Yaskawa INFORM job: OK_R2_O8B-O21B(90,0)_MPKMOK.JBI

/JOB
//NAME OK_R2_O8B-O21B(90,0)_MPKMOK
///FOLDERNAME X4
//POS
///NPOS 666,666,666,28,0,0
///TOOL 0
///POSTYPE PULSE
///PULSE
C00000=91699,-114837,-126172,-5297,65572,-69852
C00001=92194,-112793,-113721,-5907,59024,-69345
C00002=110766,-104046,-107477,-16255,62170,-62558
C00003=110766,-104165,-106515,-16351,61543,-62463
C00004=110766,-104147,-106683,-16334,61651,-62479
C00005=111036,-99665,-105018,-16294,62933,-62564
C00006=110753,-104252,-107692,-16244,62194,-62563
C00007=67116,-81864,-100907,8307,67410,-78303
C00008=67696,-81353,-98479,8065,66136,-78195
C00009=67696,-81727,-97702,8106,65471,-78242
C00010=67696,-81654,-97861,8098,65606,-78232
C00011=68924,-78441,-96430,7380,66259,-77758
C00012=67562,-81507,-99004,8124,66390,-78224
C00013=94591,-107711,-114910,-7081,62535,-68652
C00014=75177,-96078,-118139,-30635,103857,57240
C00015=71016,-101172,-117038,-29652,99603,56842
C00016=69320,-102842,-116458,-29300,97976,56637
C00017=65815,-114376,-118551,-28520,92729,56653
C00018=65815,-114603,-117718,-28482,92175,56787
C00019=65333,-115185,-120736,-28492,93393,56311
C00020=69320,-102842,-116458,-29300,97976,56637
C00021=95416,-92028,-88987,-60066,102481,86035
C00022=94783,-95327,-90301,-59871,101628,86283
C00023=95175,-93300,-89498,-59989,102155,86131
C00024=95403,-90904,-93442,-60883,104178,84663
C00025=96846,-88575,-93381,-61258,105655,84430
C00026=100267,-82342,-92970,-62384,109223,83757
C00027=98853,-105972,-123361,-35115,85568,62201
C00028=123874,-116503,-132949,-35316,93358,57662
C00029=98784,-130821,-129289,-12660,72810,27269
C00030=95442,-119682,-123188,-11300,74256,25961
C00031=89918,-115832,-119261,-9213,73142,24151
C00032=89918,-116068,-118310,-9245,72445,24204
C00033=89918,-115832,-119261,-9213,73142,24151
C00034=86534,-112000,-117975,-7848,73961,22933
C00035=89918,-115832,-119261,-9213,73142,24151
C00036=91545,-105966,-115876,-9715,76271,24462
C00037=89918,-115832,-119261,-9213,73142,24151
C00038=100559,-101270,-121421,-12879,83175,26784
C00039=103898,-109015,-126857,-14089,83070,27872
C00040=112603,-104533,-117877,-29713,115926,66306
C00041=112603,-104533,-117877,-29713,115926,66306
C00042=102787,-102282,-117268,-28859,121596,74546
C00043=102787,-103288,-115881,-28417,120387,74903
C00044=102787,-102191,-117377,-28898,121696,74514
C00045=102247,-107992,-119426,-28435,120002,74778
C00046=104853,-110239,-121572,-27980,116786,76632
C00047=123177,-144145,-129947,-26642,102859,76425
C00048=123829,-162749,-132848,-26863,92935,75206
C00049=121638,-162916,-132889,-27033,92171,74551
C00050=123829,-165003,-135169,-26874,93176,75150
C00051=112500,-101779,-108680,-28673,112161,67324
C00052=131997,-56357,-109229,4920,90907,66095
C00053=147842,-82951,-112210,34984,98309,69155
C00054=149737,-87239,-109966,34223,94635,68708
C00055=151378,-90687,-107740,33690,91394,68340
C00056=151378,-91074,-107136,33673,90915,68196
C00057=151378,-90687,-107740,33690,91394,68340
C00058=145558,-100693,-110774,34812,90892,65938
C00059=145748,-102567,-109629,34742,89434,65557
C00060=146398,-106855,-111180,34614,88141,65411
C00061=145748,-102567,-109629,34742,89434,65557
C00062=144942,-96836,-108242,34942,91483,65883
C00063=124830,-105124,-96789,55472,88700,57654
C00064=126521,-104925,-96716,55344,87736,58010
C00065=123249,-105523,-98221,55595,90026,57599
C00066=144949,-101354,-110618,34915,90771,65662
C00067=150499,-88658,-108954,33966,93222,68562
C00068=149737,-87239,-109966,34223,94635,68708
C00069=147842,-82951,-112210,34984,98309,69155
C00070=134744,-82461,-113999,23220,99839,19223
C00071=107178,-113461,-99894,5964,101445,-70182
C00072=116777,-120475,-92303,7084,92443,-67341
C00073=117649,-121004,-89231,7177,90217,-67172
C00074=117541,-124461,-90223,7160,89070,-67274
C00075=117649,-121004,-89231,7177,90217,-67172
C00076=121247,-121045,-89244,7619,89875,-65972
C00077=117649,-121004,-89231,7177,90217,-67172
C00078=120454,-123758,-93756,7530,91322,-66155
C00079=131821,-147240,-100571,7170,74455,-63187
C00080=132564,-146887,-99168,7097,73320,-62988
C00081=132564,-147261,-99594,7095,73390,-62984
C00082=116129,-123152,-95240,7006,92928,-67534
C00083=114019,-118624,-94636,6761,95050,-68140
C00084=115483,-77500,-114184,-15325,109930,-22258
C00085=107117,-124945,-135933,21570,97656,-8797
C00086=118143,-111392,-129277,15030,88270,9704
C00087=118164,-109444,-128626,15025,88847,9780
C00088=118164,-110450,-128026,15024,87989,9675
C00089=118164,-110074,-128260,15024,88315,9716
C00090=118257,-101380,-125250,15013,90827,10051
C00091=118164,-108155,-129289,15031,89881,9907
C00092=110085,-126828,-135239,17345,85673,6704
C00093=92891,-111374,-130366,26323,94899,-34453
C00094=97190,-111538,-124535,25207,90331,-33950
C00095=98877,-113015,-125031,24804,89436,-33545
C00096=97190,-111538,-124535,25207,90331,-33950
C00097=97263,-106439,-128356,25089,94874,-32878
C00098=81189,-95371,-128319,-620,93628,17487
C00099=93710,-100817,-120600,17770,81443,35553
C00100=93248,-94915,-114871,17964,81066,35345
C00101=93496,-90946,-110472,17900,80379,35326
C00102=93496,-91762,-109449,17950,79378,35179
C00103=93496,-91644,-109606,17943,79529,35199
C00104=94018,-88323,-108262,17704,80263,35482
C00105=93496,-90946,-110472,17900,80379,35326
C00106=94462,-94397,-113311,17534,80159,35616
C00107=94975,-100261,-119034,17317,80544,35841
C00108=122852,-136172,-128581,-30503,68555,-23673
C00109=143305,-96642,-110194,-35986,83923,-20153
C00110=143305,-96740,-110018,-35993,83793,-20110
C00111=143305,-97404,-108670,-36055,82835,-19796
C00112=143221,-96691,-108564,-36013,83047,-19900
C00113=142576,-91782,-106634,-35760,83882,-20426
C00114=143221,-96196,-109551,-35968,83751,-20131
C00115=92946,-121634,-121424,-16744,62834,-34226
C00116=86370,-109059,-114128,-13073,63567,-36806
C00117=86370,-109316,-113053,-13160,62794,-36714
C00118=86334,-109454,-113302,-13133,62869,-36736
C00119=87103,-105692,-111971,-13415,64077,-36592
C00120=86334,-109252,-114136,-13065,63471,-36806
C00121=121032,-150272,-131973,-30968,63431,-22949
C00122=105037,-121499,-124352,26595,83975,-43332
C00123=119038,-120466,-118045,23113,76809,-39715
C00124=125137,-115371,-113740,21293,75158,-37787
C00125=125137,-115377,-112598,21357,74498,-37908
C00126=125137,-115371,-113740,21293,75158,-37787
C00127=125247,-119622,-115037,21389,73833,-26696
C00128=125053,-112026,-112515,21239,76079,-26360
C00129=125247,-119622,-115037,21389,73833,-26696
C00130=117922,-113856,-115388,23299,78742,-39741
C00131=113283,-118224,-119490,24564,80311,-41113
C00132=130678,-94773,-121138,18217,87222,-14080
C00133=167942,-138091,-131423,-6732,80009,-27343
C00134=170575,-113227,-120751,-7300,86397,-26822
C00135=169077,-108435,-117775,-6935,86895,-27340
C00136=169077,-108900,-116810,-6936,86070,-27295
C00137=169077,-108794,-117048,-6936,86270,-27307
C00138=170304,-106542,-116256,-7229,87038,-26949
C00139=168740,-106235,-118221,-6850,88265,-27525
C00140=177701,-115390,-116622,-14957,80027,-1616
C00141=176753,-112936,-115506,-14676,80414,-1989
C00142=175630,-109912,-114469,-14334,81107,-2455
C00143=177564,-114998,-116703,-14910,80246,-1690
C00144=188009,-144692,-131667,-17931,76513,2502
C00145=152038,-126618,-128978,10588,85958,-28176
C00146=152038,-126618,-128978,10588,85958,-28176
C00147=152439,-128268,-129478,10504,85377,-28090
C00148=152439,-128687,-128060,10515,84308,-28182
C00149=152439,-128634,-128276,10513,84466,-28168
C00150=154807,-125417,-127295,9971,85207,-27314
C00151=152439,-127687,-130796,10495,86471,-28000
C00152=151563,-130369,-131601,10695,85714,-28356
C00153=164160,-102502,-129441,-9384,110509,55546
C00154=159433,-112173,-127809,-8699,104125,54469
C00155=159433,-113313,-126887,-8650,102984,54550
C00156=159433,-113125,-127052,-8657,103179,54535
C00157=157389,-116461,-128145,-8463,101945,53942
C00158=159433,-111320,-128398,-8735,104915,54410
C00159=152229,-108849,-132490,-7833,104970,48789
C00160=93963,-130535,-128792,-24722,74568,16491
C00161=90353,-119281,-117601,-23619,72522,15568
C00162=81815,-101184,-113078,-14856,80893,11838
C00163=81815,-101805,-111815,-14897,79832,11967
C00164=81815,-101566,-112336,-14880,80261,11914
C00165=81691,-96656,-110485,-14792,81580,11713
C00166=81815,-101566,-112336,-14880,80261,11914
C00167=94368,-118351,-115092,-25106,72713,8195
C00168=94368,-118242,-113051,-25259,71623,8437
C00169=92475,-116697,-112544,-24567,71499,7736
C00170=98770,-117080,-112671,-26610,73310,9747
C00171=98093,-111583,-112853,-26067,75742,17780
C00172=89023,-115119,-115343,-23068,72843,15005
C00173=90353,-119281,-117601,-23619,72522,15568
C00174=93963,-130636,-123354,-25128,71472,17166
C00175=112708,-151913,-126980,-52913,79334,-40142
C00176=108924,-145810,-121760,-52599,77119,-40924
C00177=107448,-143466,-119685,-52466,76232,-41216
C00178=107548,-140507,-116374,-52568,75966,-41003
C00179=107448,-143466,-119685,-52466,76232,-41216
C00180=124866,-69208,-71806,-74049,113649,-28483
C00181=122400,-71971,-73000,-73720,111742,-28428
C00182=124866,-69208,-71806,-74049,113649,-28483
C00183=131136,-146090,-96201,-76130,76771,-21052
C00184=127770,-141595,-95524,-76231,74990,-22221
C00185=131136,-146090,-96201,-76130,76771,-21052
C00186=112467,-159247,-111976,-60211,61283,-24397
C00187=113297,-157006,-110103,-60230,61789,-24238
C00188=113297,-157814,-110929,-60188,61836,-24279
C00189=111416,-155256,-110381,-59676,61201,-25079
C00190=114119,-159107,-112646,-60032,62541,-24296
C00191=145608,-121761,-102949,-57803,88894,-23690
C00192=146047,-120434,-101564,-57803,89067,-23542
C00193=146481,-119084,-100092,-57801,89215,-23379
C00194=146481,-119516,-101126,-57808,89444,-23539
C00195=144820,-117039,-100336,-57803,88864,-24154
C00196=147924,-121944,-103270,-57808,90363,-23296
C00197=147924,-121944,-103270,-57808,90363,-23296
C00198=137007,-126621,-110171,-48785,83769,-25153
C00199=137007,-126054,-108752,-48822,83378,-24951
C00200=137359,-125765,-109353,-48816,83916,-25050
C00201=136478,-122214,-108258,-48678,84217,-25648
C00202=137706,-129591,-111729,-48871,83766,-24798
C00203=138625,-143143,-124865,-48877,85014,-24974
C00204=98331,-144500,-124457,-41780,63547,-34680
C00205=104311,-135778,-116637,-47474,67333,-33513
C00206=104982,-134568,-114900,-47757,67380,-33183
C00207=104982,-134679,-115131,-47731,67438,-33213
C00208=102403,-135448,-115392,-47202,65913,-33778
C00209=105649,-135232,-117175,-47605,68461,-33397
C00210=103532,-169539,-136511,-48991,63433,-31812
C00211=103532,-169539,-136511,-48991,63433,-31812
C00212=22457,-72710,-105977,33427,108243,-56799
C00213=28273,-84130,-91179,49383,85325,-59450
C00214=33146,-85716,-89951,48486,81691,-58906
C00215=34224,-86775,-90401,48281,80941,-58753
C00216=34036,-86599,-90326,48317,81069,-58780
C00217=34036,-86622,-89014,48400,80515,-59063
C00218=30663,-85994,-90896,48964,83298,-59313
C00219=32844,-112560,-114598,30217,91594,-57615
C00220=32945,-106221,-111557,31487,96570,-60322
C00221=34324,-108522,-112371,31304,95486,-60091
C00222=34309,-107855,-110865,31267,94986,-60235
C00223=34309,-107970,-110045,31233,94500,-60369
C00224=34309,-107855,-110865,31267,94986,-60235
C00225=27420,-80265,-94687,41420,109338,-67363
C00226=40001,-70254,-86303,43872,85579,-70570
C00227=29252,-49748,-75503,47724,105297,-63047
C00228=36700,-141975,-135013,18885,77262,-71017
C00229=90179,-134235,-132818,-22872,80929,-49314
C00230=142804,-125519,-116198,-76046,95508,-7054
C00231=120615,-97641,-119015,-9375,90228,9949
C00232=120987,-96960,-113108,-9471,87023,10304
C00233=120613,-99917,-116962,-9368,87826,10128
C00234=121552,-104751,-117459,-9639,85780,10586
C00235=110169,-106106,-116921,-6405,83791,-7848
C00236=108950,-107035,-116988,-5812,83203,-8687
C00237=101800,-109309,-117327,-444,81272,-17192
C00238=90716,-122583,-118249,8895,71223,-28988
C00239=89439,-120853,-116474,9140,71651,-29425
C00240=89437,-130785,-128831,4407,77618,-27633
C00241=146443,-63628,-115918,3009,102570,-37934
C00242=146980,-83801,-122033,27049,110301,-76522
C00243=150856,-97054,-121393,25304,102734,-76951
C00244=152064,-99572,-120921,24941,100957,-76917
C00245=148913,-93356,-120721,25800,104620,-77205
C00246=150557,-96944,-122901,25470,103711,-76838
C00247=148071,-112807,-125003,25148,98180,-78929
C00248=146611,-117982,-126351,25207,96939,-79719
C00249=143109,-114454,-128222,25889,100648,-80164
C00250=140673,-104492,-128634,26873,106197,-79748
C00251=120599,-130072,-117206,45023,91037,-77550
C00252=120599,-129119,-114227,44983,90071,-77984
C00253=124987,-148756,-117461,44800,76699,-77028
C00254=120042,-124581,-111856,45029,90980,-77838
C00255=119368,-131507,-114599,44995,89976,-78605
C00256=124240,-148532,-116954,44871,76930,-77278
C00257=119910,-148146,-114309,45228,78097,-78816
C00258=119749,-145269,-111975,45225,78204,-78842
C00259=120598,-127933,-111142,44960,89143,-78399
C00260=120599,-129048,-114177,44983,90075,-77982
C00261=81107,-101484,-115694,-35475,102250,-71567
C00262=81518,-102603,-113057,-34270,100230,-71860
C00263=82059,-102607,-116004,-34567,101946,-72190
C00264=81374,-98102,-114013,-34658,102588,-72668
C00265=81494,-101584,-115766,-25657,104472,-80941
C00266=83161,-106402,-116658,-24816,101890,-82013
C00267=83849,-105802,-116317,-24870,102177,-81823
C00268=79384,-104922,-115530,-34104,103743,-72622
C00269=80190,-85868,-119713,-25334,110684,-45677
C00270=66991,-110384,-121517,-5418,108134,76364
C00271=56399,-121526,-132511,-11086,102541,72269
C00272=51570,-131189,-133992,-11264,103193,70513
C00273=27221,-131783,-134143,2891,99951,64006
C00274=67233,-108188,-115958,-5335,105866,76549
C00275=66897,-113678,-118543,-5308,104619,76489
C00276=41481,-133217,-133850,-4573,100163,77286
C00277=41042,-124946,-131371,-1999,105337,72535
C00278=41185,-117707,-128794,2243,111064,68602
C00279=63882,-97812,-119916,-5442,123090,74934
C00280=71451,-102497,-120744,-3949,121646,77876
C00281=87989,-107726,-120992,-589,118665,84191
C00282=84930,-119629,-129782,1888,113436,83486
C00283=84729,-121080,-124653,-20914,107476,65948
C00284=95444,-112372,-114390,-31511,111945,67927
C00285=67316,-107916,-115567,9495,105572,72905
C00286=66579,-114256,-118448,9402,104190,72540
C00287=98021,-122686,-116586,-31197,106837,67491
C00288=98017,-122619,-115764,-31114,106429,67606
C00289=102197,-111658,-121490,-32833,115802,66493
C00290=86428,-100957,-127747,-22004,113840,67454
C00291=53800,-100419,-127772,3487,91936,72900
C00292=55487,-108533,-124083,2963,85444,73257
C00293=54649,-108835,-123171,3222,84756,72973
C00294=54376,-102036,-122875,3303,88076,72973
C00295=53684,-106892,-125333,3516,87122,72731
C00296=51776,-104500,-121658,4102,86181,72100
C00297=52810,-105662,-121978,3788,85735,72414
C00298=53695,-106380,-122097,3513,85396,72684
C00299=53834,-105518,-125265,3470,87779,72796
C00300=58883,-114751,-131257,1913,86567,74352
C00301=99205,-132197,-126076,-29274,71590,-12900
C00302=100538,-139639,-126656,-10769,67376,-15479
C00303=99890,-133434,-123018,-10459,68226,-15794
C00304=121557,-117112,-114069,-35409,80373,-6489
C00305=120930,-112739,-113965,-35102,81919,-7240
C00306=105243,-128809,-121738,-14815,71739,-11607
C00307=119667,-108803,-109812,-34841,80971,-7453
C00308=133655,-88048,-99327,-37721,90153,-4837
C00309=135782,-84357,-97373,-38144,91605,-4481
C00310=120608,-113488,-111079,-35194,80005,-6758
C00311=120913,-113610,-118761,-34960,83981,-7901
C00312=60517,-140064,-128137,5523,60575,-30169
C00313=76507,-136356,-126633,15520,62258,-37847
C00314=93877,-119513,-106917,30240,50522,-43245
C00315=93872,-118929,-104978,30616,49748,-43511
C00316=96675,-114118,-101851,28706,49234,-42274
C00317=91867,-119287,-104388,32007,50022,-44430
C00318=93165,-122201,-105305,31680,48734,-44232
C00319=96575,-112981,-98851,29299,48158,-42676
C00320=93870,-118064,-102441,31104,48784,-43850
C00321=93875,-120519,-110719,29525,52112,-42724
C00322=103713,-78156,-110673,21781,86340,-9498
C00323=103152,-115418,-123402,33822,74617,14862
C00324=124928,-109292,-104782,36694,51003,34659
C00325=125167,-95419,-100236,32669,59273,37861
C00326=127956,-93582,-99677,30982,58761,38938
C00327=134682,-88838,-97728,26765,57595,41519
C00328=133665,-87494,-99701,26855,59621,41625
C00329=106977,-98611,-100510,42515,63569,28708
C00330=121083,-121277,-109751,27112,45366,37764
C00331=121016,-120747,-110300,26892,45934,37909
C00332=106032,-97399,-100028,43035,64662,28283
C00333=106877,-98272,-101332,41419,65450,27289
C00334=120722,-118203,-110949,26093,49137,36520
C00335=96719,-133488,-134181,17465,82071,-6810
C00336=88208,-121632,-130599,22903,100986,-52847
C00337=98918,-140805,-130229,21227,89577,-51155
C00338=101812,-147602,-128384,21006,84502,-50993
C00339=106194,-98373,-112810,20835,98142,-47084
C00340=98278,-109583,-120915,21720,99368,-49630
C00341=124341,-131813,-131636,-11198,92459,43971
C00342=121621,-98285,-117221,-11998,109073,41436
C00343=120829,-102076,-117837,-11863,107428,41331
C00344=120902,-107261,-118230,-11233,92587,42752
C00345=120747,-112603,-128286,-11278,95948,42397
C00346=120609,-111837,-120554,-26049,67413,-30439
C00347=127530,-87243,-106087,-27145,76004,-54708
C00348=127855,-101263,-105463,-29286,62195,-54682
C00349=120275,-109775,-109691,-27025,62250,-29299
C00350=120607,-113891,-112343,-27298,61925,-29076
C00351=124642,-99236,-105815,-26754,63612,-56360
C00352=124642,-99246,-105774,-26761,63584,-56353
C00353=119464,-101431,-106692,-24188,61661,-57984
C00354=117484,-140120,-126379,6353,63040,-48502
C00355=118425,-101447,-120931,2723,88548,-49569
C00356=118902,-98684,-118530,2584,88476,-49421
C00357=112623,-148045,-125948,8820,59190,-50637
C00358=91638,-143197,-119722,29396,63714,-58185
C00359=84683,-155167,-127701,31711,65172,-60743
C00360=119412,-103833,-118895,8159,86026,-48306
C00361=120645,-103801,-122240,-18363,79401,-46323
C00362=120596,-133604,-113690,-59811,77806,-45056
C00363=120595,-131656,-109787,-60053,77075,-44491
C00364=112007,-157167,-113694,-61825,56110,-45689
C00365=121130,-127010,-106775,-60003,77686,-44610
C00366=122155,-131356,-109255,-60198,77961,-44142
C00367=113123,-156836,-112841,-62124,56631,-45300
C00368=117315,-158239,-111132,-63346,58407,-43675
C00369=117620,-158110,-110791,-63433,58531,-43555
C00370=120595,-130364,-107240,-60219,76607,-44125
C00371=120595,-136323,-119613,-59458,78987,-45957
C00372=120692,-96649,-118672,-32375,84269,-53596
C00373=120600,-118120,-97579,-10821,96522,-62450
C00374=120599,-116060,-93092,-10778,94848,-62304
C00375=104457,-125932,-94017,-2632,84881,-67774
C00376=120596,-116950,-93034,-10767,94362,-62263
C00377=120597,-112553,-90859,-10788,95268,-62342
C00378=105526,-126673,-94317,-2582,84718,-67411
C00379=113928,-128065,-94704,-2162,84487,-64572
C00380=114617,-128092,-94646,-2128,84458,-64339
C00381=120599,-116103,-93113,-10778,94839,-62304
C00382=120600,-118165,-97601,-10821,96512,-62449
C00383=119173,-110104,-84650,17860,100738,-60179
C00384=121454,-109687,-81979,18272,98871,-59635
C00385=119205,-107046,-82886,17903,101194,-60099
C00386=117500,-110311,-84228,17454,100749,-60784
C00387=120748,-108893,-80959,18105,98817,-59897
C00388=118360,-105961,-77958,17548,99011,-60728
C00389=118025,-105641,-77691,17472,99083,-60836
C00390=119269,-105795,-90384,16222,103319,-56958
C00391=119250,-107896,-92223,16223,103373,-56958
C00392=120631,-120794,-104165,-3096,101272,12664
C00393=93681,-116199,-92959,-21871,86687,63192
C00394=93682,-114281,-89064,-21892,85374,63431
C00395=93994,-112402,-84988,-21921,84020,63792
C00396=94896,-115380,-88949,-21880,85105,63922
C00397=94330,-111162,-87177,-21872,85957,63561
C00398=97211,-111244,-82023,-21869,83727,65014
C00399=93688,-114747,-90039,-16462,83105,67478
C00400=98020,-112989,-101813,-16504,91812,67842
C00401=120691,-83893,-117951,-31034,76795,-369
C00402=109337,-117271,-103204,-33165,32410,-56709
C00403=108598,-118256,-100577,-34319,30336,-56092
C00404=117114,-110300,-87677,-73061,48036,-44279
C00405=120810,-118458,-98421,-46795,34964,-49508
C00406=120898,-120190,-100727,-46315,35380,-49771
C00407=99913,-110179,-102111,725,37211,-74486
C00408=94755,-104895,-101725,12221,42726,-80312
C00409=96213,-105350,-101945,10935,42423,-79630
C00410=99969,-107364,-102297,7624,41187,-77884
C00411=117793,-111917,-101498,-9811,38580,-68613
C00412=116786,-129112,-111653,-9356,35906,-68838
C00413=120602,-119646,-106124,-23770,35755,-64006
C00414=120572,-164631,-130559,-29498,28477,-60984
C00415=59378,-79993,-117615,-20992,104349,-50993
C00416=59534,-83013,-114526,-20694,101146,-50372
C00417=77175,-58036,-93366,-41069,112824,-50974
C00418=58372,-87022,-114306,-20279,98825,-50352
C00419=59444,-82986,-114089,-20654,100887,-50356
C00420=65092,-37882,-81766,-40150,110396,-55003
C00421=48464,-53437,-100454,-18522,104822,-54763
C00422=48227,-49677,-102991,-18845,108096,-55363
C00423=80679,-104141,-125686,-9644,102744,-40683
C00424=118067,-125720,-131229,18141,88550,-23791
C00425=119196,-107213,-115583,19115,87640,-23373
C00426=121699,-105262,-112483,19242,86972,-21598
C00427=117080,-103991,-114571,20230,89872,-22719
C00428=116066,-108230,-114829,20428,88214,-23347
C00429=122381,-105719,-113331,9069,82450,-8912
C00430=126696,-108373,-114128,6771,80419,-568
C00431=142779,-103158,-112224,-8798,82570,16248
C00432=121247,-109622,-114889,-13373,78296,4610
C00433=134056,-113869,-113144,21646,71523,-28395
C00434=136867,-109744,-110142,20577,71068,-27434
C00435=132204,-114603,-112784,22383,71453,-29101
C00436=133799,-109730,-110978,21650,72329,-28339
C00437=136032,-108951,-108189,20981,70531,-27843
C00438=134059,-113755,-114816,16878,74881,-27676
C00439=134057,-113222,-117239,16761,76575,-27439
C00440=134085,-122795,-122723,-12562,74454,19579
C00441=134084,-123052,-120179,-12662,72796,19752
C00442=133873,-119304,-117433,-12589,72993,19657
C00443=134370,-128050,-120849,-12910,70736,20076
C00444=135935,-124649,-119997,-13370,72179,20478
C00445=136397,-117290,-114619,-14497,73201,21549
C00446=134086,-122982,-121548,-14244,80726,12740
C00447=134086,-122460,-124273,-14187,82615,12522
C00448=124281,-111431,-128342,-21366,88313,-4883
C00449=101088,-90789,-125448,-21651,85172,-29871
C00450=93918,-104964,-136200,-23440,91622,-46043
C00451=93920,-124128,-120530,-24248,73694,-42461
C00452=94513,-120070,-115912,-24522,73175,-42126
C00453=94160,-120648,-118787,-24248,74418,-42523
C00454=93561,-129068,-120517,-24441,71260,-42079
C00455=94538,-119909,-115716,-24538,73146,-42109
C00456=94540,-119894,-116072,-24510,73350,-42158
C00457=85322,-114853,-114435,-21214,72301,-45396
C00458=84866,-114469,-114315,-21036,72300,-45564
C00459=93972,-122221,-127126,-23802,78331,-43399
C00460=95212,-124771,-130616,-25606,80781,-41793
C00461=95212,-124771,-130616,-25606,80781,-41793
C00462=95212,-124771,-130616,-25606,80781,19677
C00463=87283,-86668,-106269,-24673,86609,15333
C00464=87767,-89166,-101962,-24913,83160,16227
C00465=89149,-106557,-109914,-23947,75942,18492
C00466=123530,-75295,-101290,-33091,96563,25932
C00467=124593,-95792,-102495,-38038,80779,30244
C00468=124599,-96235,-97339,-38396,78076,31222
C00469=128762,-97835,-105146,-39063,83045,31166
C00470=66215,-117666,-119596,4204,73122,9588
C00471=69871,-90679,-106158,-3816,81936,13325
C00472=47201,-74326,-98737,19988,93542,-10859
C00473=75658,-90208,-105781,13162,84947,-3532
C00474=78119,-89100,-105460,11903,84687,-2157
C00475=102348,-78970,-101207,6657,85431,3272
C00476=89814,-57389,-91066,21641,98724,-12051
C00477=83302,-63123,-101501,23427,103509,-13270
C00478=82075,-65501,-105338,23833,104858,-13394
C00479=96888,-120810,-128549,-8566,82721,50200
C00480=107399,-123550,-122639,-19719,77762,53336
C00481=105987,-126908,-125537,-19297,77487,52876
C00482=105708,-123198,-122518,-19211,77470,52780
C00483=100131,-75267,-104498,-17084,89205,49156
C00484=101170,-74384,-108530,-17462,92208,49062
C00485=110716,-78612,-119218,-29200,98920,-42289
C00486=6723,-78612,-119218,-29200,98920,-42289
C00487=-26149,-48715,-68613,7646,64296,-87864
C00488=37227,-117034,-86146,32359,44380,-13289
C00489=81285,-37438,-50804,21684,56778,30387
C00490=80438,9168,-10717,26405,57944,34662
C00491=78877,19020,-1177,27491,57718,33926
C00492=78745,21063,1089,27662,57453,33795
C00493=78745,21075,2041,27832,56937,33652
C00494=78745,21070,1795,27788,57069,33689
C00495=78800,22355,3015,27785,56971,33687
C00496=78880,19396,-683,27521,57617,33902
C00497=80581,13500,-4347,26804,56376,34308
C00498=80587,8416,-11814,26244,58158,34782
C00499=112932,28382,-4139,2581,62718,48966
C00500=146242,42258,30664,-20511,46292,62528
C00501=144329,45415,35078,-19510,44794,61921
C00502=144875,45947,36603,-20134,44299,62311
C00503=144875,46417,38447,-20453,43460,62510
C00504=144875,46350,38193,-20408,43574,62483
C00505=144568,46514,38370,-20191,43475,62348
C00506=144875,46000,36820,-20170,44200,62334
C00507=149300,7617,-13124,-20056,55660,61959
C00508=110214,39149,6684,-28287,96687,48296
C00509=93936,66202,45488,-26008,82562,45514
C00510=94391,67020,49295,-26174,80971,46039
C00511=94391,67246,50410,-26209,80457,46153
C00512=94391,67082,49603,-26185,80829,46070
C00513=95479,65713,48782,-26351,80993,46446
C00514=95018,65028,47987,-26279,80969,46276
C00515=95450,66206,49577,-26361,80771,46485
C00516=95450,65446,45347,-26245,82765,46037
C00517=94280,85401,67758,-24935,85608,70946
C00518=95136,79608,63100,-27514,83348,85198
C00519=95290,77489,60518,-27509,83845,85139
C00520=95109,79640,61859,-27482,84035,85026
C00521=96461,73500,53539,-20575,81665,48796
C00522=96145,75246,60941,-20725,78149,49286
C00523=96145,75860,63054,-20793,77228,49448
C00524=96389,75627,62622,-20821,77426,49500
C00525=95545,75058,61940,-20687,77334,49209
C00526=95970,73750,56673,-20593,79851,48927
C00527=97227,50986,24249,-20554,87918,48006
C00528=115023,23375,-7873,-26249,84597,51324
C00529=148711,-61590,-86342,-17909,64527,60132
C00530=122925,-41472,-107688,-1595,85037,50935
C00531=122274,54028,61959,-1512,43476,35052
C00532=122041,57255,48823,-1076,55606,31980
C00533=120248,71316,67884,-205,51086,31263
C00534=120244,68458,65853,-201,50866,31262
C00535=120244,69525,68499,-204,49787,31263
C00536=120244,69345,68062,-204,49964,31263
C00537=120041,71390,70509,-98,49510,31175
C00538=120243,67493,64509,-200,51199,31260
C00539=112329,62453,61247,5556,54103,20424
C00540=113214,68347,70966,5362,51097,20637
C00541=112423,63328,63484,5579,53174,20413
C00542=112135,65306,64495,5681,53586,20316
C00543=114303,70753,73426,4015,51411,20260
C00544=116065,74970,78829,4033,49561,21714
C00545=115368,69103,69060,4259,52532,21613
C00546=115921,59846,55216,3823,56258,21985
C00547=122274,54028,61959,-1512,43476,35052
C00548=122925,-41472,-107688,-1595,85037,50935
C00549=148711,-64912,-77096,-19175,57496,385
C00550=87963,22704,-863,-14505,81421,-75380
C00551=82398,26437,15461,-20580,61726,-74959
C00552=79758,26511,15534,-19458,61075,-75904
C00553=79590,7840,-1747,-19205,62020,-76144
C00554=82428,7690,-1878,-20408,62708,-75135
C00555=82725,7077,-4572,-20305,64043,-75266
C00556=85834,18050,6851,-21811,63534,-73932
C00557=93318,16641,24413,-51343,49736,-63367
C00558=93949,17768,19147,-42943,61010,-68605
C00559=93013,19529,17580,-41735,62477,-69710
C00560=89531,18173,-4575,-15569,81534,-74809
C00561=83245,47983,25939,-9273,90468,-77050
C00562=83005,68520,52515,-10136,92332,-77290
C00563=81919,51967,31879,-9150,88730,-77372
C00564=81934,49381,27809,-9155,89894,-77452
C00565=82786,64696,48407,-13279,91233,-77339
C00566=82019,48878,26914,-9164,90191,-77445
C00567=88083,33116,10426,-9703,92913,-75595
C00568=86953,39537,8218,-12835,90174,-73057
C00569=81396,82023,55882,-32097,38956,-53680
C00570=81190,90464,69323,-34749,35562,-52175
C00571=81786,101118,84455,-38671,32706,-50061
C00572=81108,93968,73693,-35396,34795,-51817
C00573=81117,90662,70751,-35312,34890,-51864
C00574=80128,100963,84245,-37069,32021,-50912
C00575=79314,90463,69327,-33002,34812,-53080
C00576=79483,82000,55858,-30378,38255,-54553
C00577=109961,31343,-14451,-13674,84826,-9825
C00578=157666,-56380,-75230,-23755,62771,63830
C00579=122925,-41472,-107688,-1595,85037,50935
C00580=122274,54028,61959,-1512,43476,35052
C00581=106492,37397,54240,-2185,50844,9950
C00582=113507,46568,52063,-21056,60301,-577
C00583=112968,55940,65611,-21671,56871,-98
C00584=113074,61965,75196,-22405,54295,513
C00585=113067,57215,68339,-21946,55944,142
C00586=112759,58823,68838,-21733,56347,-74
C00587=115594,68450,82911,-23479,53668,1745
C00588=114945,60069,70362,-22403,56644,781
C00589=115521,50177,56014,-21714,60281,248
C00590=122274,54028,61959,-1512,43476,35052
C00591=123169,-59815,-117332,-1745,81551,51041
C00592=151982,-78435,-94523,-20407,61819,61824
C00593=151982,-78435,-94523,-20407,61819,-25376
C00594=134688,6231,-23564,-20522,94268,-37191
C00595=115943,62792,41458,-21315,104693,-45869
C00596=114029,67421,50572,-21383,103633,-46383
C00597=113789,72753,60871,-20342,102004,-46157
C00598=121400,68431,53573,-20011,104381,-43747
C00599=121752,65544,48943,-20095,105754,-43852
C00600=111850,68967,56387,-20759,102286,-46928
C00601=115399,52393,31818,-20910,109375,-46865
C00602=124095,50320,22708,-12675,91472,-6833
C00603=118971,49257,27765,-7041,74456,12013
C00604=118344,55145,37167,-6948,71660,11954
C00605=121691,77951,64253,-13726,74224,16877
C00606=118100,57432,39652,-6887,71288,11889
C00607=118438,55380,38603,-7006,70911,12031
C00608=120302,74221,59820,-13402,74782,16316
C00609=121648,62314,45296,-16341,75480,15894
C00610=122678,56843,36157,-16407,78391,15868
C00611=150584,-71485,-91286,-19317,62987,61079
C00612=123050,-50840,-112823,-1671,83386,50986
C00613=115744,32670,26267,2188,54498,32210
C00614=103599,34577,51597,-1741,50803,1907
C00615=103485,36027,47218,-1621,54239,1804
C00616=104787,41655,55707,-8390,53564,5846
C00617=103440,38491,49687,-1609,53985,1789
C00618=103682,37013,49483,-1714,53356,1898
C00619=109485,48740,63382,-11917,54003,11492
C00620=107897,40852,51906,-12631,57379,14673
C00621=108788,40242,57118,-13430,54084,15447
C00622=122274,54028,61959,-1512,43476,35052
C00623=122925,-41472,-107688,-1595,85037,50935
C00624=148711,-64771,-77902,-19060,58035,61239
C00625=141930,24245,-13757,-17037,93950,-6277
C00626=132421,69326,40341,-15933,104552,-53546
C00627=127843,72860,44976,-16143,102664,-54937
C00628=127479,95684,77579,-21551,102467,-55073
C00629=123966,73267,47056,-16275,100870,-56082
C00630=124331,70889,42989,-16346,102176,-56130
C00631=125868,89416,69574,-21985,103631,-55895
C00632=126217,68327,39621,-16307,103273,-55604
C00633=126051,70827,38573,-16479,105096,-55916
C00634=136631,70064,39172,-19099,86104,19657
C00635=135438,74299,47124,-18933,83255,19683
C00636=134979,79038,54861,-18933,80945,19882
C00637=134970,76095,49205,-18856,82809,19586
C00638=135406,74025,47966,-18948,82624,19770
C00639=133572,73844,48656,-18621,81710,19257
C00640=133939,69065,40918,-18618,83988,19040
C00641=135132,65055,33319,-18804,86739,19035
C00642=153194,47181,13376,-14776,85463,24597
C00643=151929,50472,19874,-14503,83006,24461
C00644=150210,50397,22217,-14109,81274,24075
C00645=152015,50489,21062,-14543,82321,24570
C00646=151435,52018,21490,-14383,82726,24324
C00647=150867,57430,30163,-14317,80149,24431
C00648=150602,54025,23778,-14183,82219,24099
C00649=154930,55090,22038,-15225,84547,25295
C00650=129519,59293,25405,-9085,104952,-46428
C00651=132629,59775,29887,-8641,103814,-47917
C00652=130987,64624,38903,-4811,101881,-55886
C00653=137538,62472,33316,-8375,103603,-46193
C00654=137071,64325,36692,-8355,102443,-46276
C00655=130203,72205,47872,-4828,100215,-56089
C00656=129031,66361,39814,-6448,101513,-53947
C00657=135480,49748,14386,-7583,108745,-49839
C00658=138083,40993,19031,-10964,76619,20362
C00659=146399,54791,36852,-13432,74072,23552
C00660=141133,53137,37638,-12088,71937,21890
C00661=146486,55146,38421,-13505,73324,23667
C00662=145946,56601,38797,-13329,73737,23427
C00663=141178,60165,45502,-12183,70755,22025
C00664=141841,45130,25495,-12091,75333,21800
C00665=152489,39248,15320,-14733,80233,24982
BC00000=369143,285250,1075139
BC00001=369143,285250,1075139
BC00002=369143,285250,1075139
BC00003=369143,285250,1075139
BC00004=369143,285250,1075139
BC00005=369143,285250,1075139
BC00006=369143,285250,1075139
BC00007=369143,285250,1075139
BC00008=369143,285250,1075139
BC00009=369143,285250,1075139
BC00010=369143,285250,1075139
BC00011=369143,285250,1075139
BC00012=369143,285250,1075139
BC00013=369143,285250,1075139
BC00014=304369,328121,1075139
BC00015=304369,328121,1075139
BC00016=304369,328121,1075139
BC00017=304369,328121,1075139
BC00018=304370,328120,1075138
BC00019=304369,328121,1075139
BC00020=304369,328121,1075139
BC00021=304369,328121,1075139
BC00022=304369,328121,1075139
BC00023=304369,328121,1075139
BC00024=304369,328121,1075139
BC00025=304369,328121,1075139
BC00026=304369,328121,1075139
BC00027=288312,290563,1075139
BC00028=281943,275865,1075139
BC00029=267232,241912,1075139
BC00030=267232,241912,1075139
BC00031=267232,241912,1075139
BC00032=267232,241912,1075139
BC00033=267232,241912,1075139
BC00034=267232,241912,1075139
BC00035=267232,241912,1075139
BC00036=267232,241912,1075139
BC00037=267232,241912,1075139
BC00038=267232,241912,1075139
BC00039=267232,241912,1075139
BC00040=235633,192426,1075139
BC00041=251897,204810,1058528
BC00042=252581,192012,1058528
BC00043=252581,192012,1058528
BC00044=252581,192012,1058528
BC00045=252581,192012,1058528
BC00046=252581,192012,1058528
BC00047=252581,192012,1058528
BC00048=252581,192012,1058528
BC00049=252581,192012,1058528
BC00050=252581,192012,1058528
BC00051=235633,249567,1075139
BC00052=303430,339929,1075139
BC00053=349686,261376,1075139
BC00054=349686,261376,1075139
BC00055=349686,261376,1075139
BC00056=349686,261376,1075139
BC00057=349686,261376,1075139
BC00058=349686,261376,1075139
BC00059=349686,261376,1075139
BC00060=349686,261376,1075139
BC00061=349686,261376,1075139
BC00062=349686,261376,1075139
BC00063=349686,261376,1075139
BC00064=349686,261376,1075139
BC00065=349686,261376,1075139
BC00066=349686,261376,1075139
BC00067=349686,261376,1075139
BC00068=349686,261376,1075139
BC00069=349686,261376,1075139
BC00070=320394,326243,1075159
BC00071=271050,384476,1075193
BC00072=271050,384476,1075193
BC00073=271051,384476,1075189
BC00074=271051,384476,1075189
BC00075=271051,384476,1075189
BC00076=271051,384476,1075189
BC00077=271051,384476,1075189
BC00078=271051,384476,1075189
BC00079=271051,384476,1075189
BC00080=271051,384476,1075189
BC00081=271051,384476,1075189
BC00082=271050,384476,1075193
BC00083=271050,384476,1075193
BC00084=239792,334493,1075164
BC00085=370673,321740,1037212
BC00086=370673,342400,1005362
BC00087=370673,342400,1005362
BC00088=370673,342400,1005362
BC00089=370673,342400,1005362
BC00090=370673,342400,1005362
BC00091=370673,342400,1005362
BC00092=370673,342400,1005362
BC00093=370673,342400,1005362
BC00094=370673,342400,1005362
BC00095=370673,342400,1005362
BC00096=370673,342400,1005362
BC00097=370160,342160,1005589
BC00098=209829,261158,1075139
BC00099=213419,253004,1075139
BC00100=213419,253004,1075139
BC00101=213419,253004,1075139
BC00102=213419,253004,1075139
BC00103=213419,253004,1075139
BC00104=213419,253004,1075139
BC00105=213419,253004,1075139
BC00106=213419,253004,1075139
BC00107=213419,253004,1075139
BC00108=89246,224121,1075139
BC00109=89246,224121,1075139
BC00110=89246,224121,1075139
BC00111=89246,224121,1075139
BC00112=89246,224121,1075139
BC00113=89246,224121,1075139
BC00114=89246,224121,1075139
BC00115=89246,224121,1075139
BC00116=89246,224121,1075139
BC00117=89246,224121,1075139
BC00118=89246,224121,1075139
BC00119=89246,224121,1075139
BC00120=89246,224121,1075139
BC00121=89246,224121,1075139
BC00122=154797,231156,1075139
BC00123=154797,231156,1075139
BC00124=154797,231156,1075139
BC00125=154797,231156,1075139
BC00126=154797,231156,1075139
BC00127=154797,231156,1075139
BC00128=154797,231156,1075139
BC00129=154797,231156,1075139
BC00130=154797,231156,1075139
BC00131=154797,231156,1075139
BC00132=146041,254218,1075139
BC00133=134978,219294,1075139
BC00134=129971,219294,1075139
BC00135=129971,219294,1075139
BC00136=129971,219294,1075139
BC00137=129971,219294,1075139
BC00138=129971,219294,1075139
BC00139=129971,219294,1075139
BC00140=129971,219294,1075139
BC00141=129971,219294,1075139
BC00142=129971,219294,1075139
BC00143=129971,219294,1075139
BC00144=129971,219294,1075139
BC00145=129971,273892,1075139
BC00146=123663,276164,1045788
BC00147=122637,276612,1036919
BC00148=122637,276612,1036919
BC00149=122637,276612,1036919
BC00150=122637,276612,1036919
BC00151=122637,276612,1036919
BC00152=122637,276612,1036919
BC00153=122637,276612,1036919
BC00154=122637,276612,1036919
BC00155=122637,276612,1036919
BC00156=122637,276612,1036919
BC00157=122637,276612,1036919
BC00158=122637,276612,1036919
BC00159=124638,273047,1041880
BC00160=141157,261252,1075139
BC00161=141157,261252,1075139
BC00162=141157,261252,1075139
BC00163=141157,261252,1075139
BC00164=141157,261252,1075139
BC00165=141157,261252,1075139
BC00166=141157,261252,1075139
BC00167=141157,261252,1075136
BC00168=141157,261252,1075136
BC00169=141157,261252,1075136
BC00170=141157,261252,1075136
BC00171=141157,261252,1075139
BC00172=141157,261252,1075139
BC00173=141157,261252,1075139
BC00174=141157,261252,1075139
BC00175=344298,346637,1075139
BC00176=344298,346637,1075139
BC00177=344298,346637,1075139
BC00178=344298,346637,1075139
BC00179=344298,346637,1075139
BC00180=344298,346637,1075139
BC00181=344298,346637,1075139
BC00182=344298,346637,1075139
BC00183=344298,346637,1075139
BC00184=344298,346637,1075139
BC00185=344298,346637,1075139
BC00186=344298,346637,1075139
BC00187=344298,346637,1075139
BC00188=344298,346637,1075139
BC00189=344298,346637,1075139
BC00190=344298,346637,1075139
BC00191=344298,346637,1075139
BC00192=344298,346637,1075139
BC00193=344298,346637,1075139
BC00194=344298,346637,1075139
BC00195=344298,346637,1075139
BC00196=344298,346637,1075139
BC00197=305690,324653,1075139
BC00198=305690,324653,1075139
BC00199=305690,324653,1075139
BC00200=305690,324653,1075139
BC00201=305690,324653,1075139
BC00202=305690,324653,1075139
BC00203=305690,324653,1075139
BC00204=305690,324653,1075139
BC00205=305690,324653,1075139
BC00206=305690,324653,1075139
BC00207=305690,324653,1075139
BC00208=305690,324653,1075139
BC00209=305690,324653,1075139
BC00210=305690,324653,1075139
BC00211=391454,377155,1075139
BC00212=391454,377155,1075139
BC00213=391454,377155,1075139
BC00214=391454,377155,1075139
BC00215=391454,377155,1075139
BC00216=391454,377155,1075139
BC00217=391454,377155,1075139
BC00218=391454,377155,1075139
BC00219=391454,377155,1075139
BC00220=391454,377155,1075139
BC00221=391454,377155,1075139
BC00222=391454,377155,1075139
BC00223=391454,377155,1075139
BC00224=391454,377155,1075139
BC00225=391453,377155,1075138
BC00226=391453,377155,1075138
BC00227=391454,377155,1075139
BC00228=391454,377155,1075139
BC00229=374557,368183,1075139
BC00230=283294,319724,1075139
BC00231=214088,291593,1075139
BC00232=217298,284602,1075136
BC00233=217299,284603,1075139
BC00234=217299,284603,1075139
BC00235=217298,284602,1075136
BC00236=217298,284602,1075136
BC00237=217298,284602,1075133
BC00238=217297,284603,1075129
BC00239=217297,284603,1075129
BC00240=216649,284539,1075130
BC00241=305960,297188,1058377
BC00242=324560,244674,1036586
BC00243=324560,244674,1036586
BC00244=324560,244674,1036586
BC00245=324560,244674,1036586
BC00246=324560,244674,1036586
BC00247=324560,244674,1036586
BC00248=324560,244674,1036586
BC00249=324560,244674,1036586
BC00250=324560,244674,1036586
BC00251=339829,244579,1075139
BC00252=334450,247303,1075139
BC00253=332299,248392,1075139
BC00254=332299,248392,1075139
BC00255=332299,248392,1075139
BC00256=332299,248392,1075139
BC00257=332299,248392,1075139
BC00258=332299,248392,1075139
BC00259=338969,248286,1075139
BC00260=344348,245562,1075139
BC00261=139995,218400,1075139
BC00262=141091,220907,1075139
BC00263=141091,220907,1075139
BC00264=141091,220907,1075139
BC00265=152171,222661,1075139
BC00266=151559,222081,1075132
BC00267=151559,222081,1075132
BC00268=141059,209205,1075139
BC00269=159708,237485,1075139
BC00270=246751,249525,1075139
BC00271=245595,202156,1075139
BC00272=273914,202156,1075139
BC00273=277230,202156,1075139
BC00274=245133,253819,1075139
BC00275=245133,253819,1075139
BC00276=277230,202156,1075139
BC00277=277230,202156,1075139
BC00278=277230,202156,1075139
BC00279=277230,202156,1075139
BC00280=277230,202156,1075139
BC00281=277230,202156,1075139
BC00282=277230,202156,1075139
BC00283=231262,184184,1075139
BC00284=231262,184184,1075139
BC00285=289900,285131,1075139
BC00286=289900,285131,1075139
BC00287=231262,184184,1075139
BC00288=231262,184184,1075139
BC00289=231262,184184,1075139
BC00290=267679,235233,1075139
BC00291=343240,341153,1075139
BC00292=344095,341334,1075139
BC00293=344218,341360,1075139
BC00294=344218,341360,1075139
BC00295=344218,341360,1075139
BC00296=348355,343666,1075139
BC00297=359572,349952,1075139
BC00298=363699,352275,1075139
BC00299=363419,352216,1075139
BC00300=363419,352216,1075139
BC00301=263777,330087,1075139
BC00302=302548,333700,1075139
BC00303=302548,333700,1075139
BC00304=268346,323394,1075139
BC00305=268346,323394,1075139
BC00306=279343,320698,1075133
BC00307=264650,321320,1075136
BC00308=264650,321320,1075136
BC00309=264650,321320,1075136
BC00310=241341,310889,1075139
BC00311=238077,315670,1075139
BC00312=238077,315670,1075139
BC00313=307250,356623,1075139
BC00314=353410,383952,1075139
BC00315=349816,377904,1075139
BC00316=348379,375484,1075139
BC00317=348379,375484,1075139
BC00318=348379,375484,1075139
BC00319=348379,375484,1075139
BC00320=349814,377891,1075139
BC00321=353407,383939,1075139
BC00322=302706,337798,1075139
BC00323=251047,291951,1075139
BC00324=251497,257349,1075138
BC00325=251497,257349,1075138
BC00326=251497,257349,1075138
BC00327=251497,257349,1075138
BC00328=251497,257349,1075138
BC00329=211375,253814,1075136
BC00330=211374,253814,1075139
BC00331=211374,253814,1075139
BC00332=206696,252912,1075139
BC00333=124253,237017,1075136
BC00334=119410,238478,1075139
BC00335=61845,243405,1075139
BC00336=69065,219693,1065143
BC00337=69141,285139,1065143
BC00338=69141,285139,1065143
BC00339=69141,285139,1065143
BC00340=69141,285139,1065143
BC00341=69141,285139,1065143
BC00342=69141,285139,1065143
BC00343=69141,285139,1065143
BC00344=69141,285139,1065143
BC00345=69141,285139,1065143
BC00346=211083,265895,1075139
BC00347=211388,260435,1075139
BC00348=211388,260435,1075139
BC00349=211510,258251,1075139
BC00350=211510,258251,1075139
BC00351=211388,260435,1075139
BC00352=211388,260435,1075139
BC00353=211388,260435,1075139
BC00354=262640,231803,1075139
BC00355=262640,231803,1075139
BC00356=262640,231803,1075139
BC00357=262640,231803,1075139
BC00358=262640,231803,1075139
BC00359=262640,231803,1075139
BC00360=279577,236209,1075139
BC00361=226569,246114,1075139
BC00362=139868,198005,1075139
BC00363=144589,196993,1075139
BC00364=146477,196588,1075139
BC00365=146477,196588,1075139
BC00366=146477,196588,1075139
BC00367=146477,196589,1075138
BC00368=146477,196588,1075139
BC00369=146477,196588,1075139
BC00370=140485,199082,1075139
BC00371=135765,200094,1075139
BC00372=192409,368654,1075139
BC00373=235005,390046,1075139
BC00374=234294,393257,1075139
BC00375=234010,394542,1075137
BC00376=234010,394542,1075139
BC00377=234010,394542,1075139
BC00378=234010,394542,1075137
BC00379=234010,394542,1075137
BC00380=234010,394542,1075137
BC00381=225235,393242,1075139
BC00382=225946,390031,1075139
BC00383=290301,380894,1075139
BC00384=288616,382418,1075139
BC00385=288616,382418,1075139
BC00386=288616,382418,1075139
BC00387=288616,382418,1075139
BC00388=288616,382418,1075139
BC00389=288616,382418,1075139
BC00390=291524,385023,1075139
BC00391=291524,385023,1075139
BC00392=238695,387513,1075169
BC00393=160865,383662,1075193
BC00394=164325,387264,1075193
BC00395=165709,388705,1075193
BC00396=165709,388705,1075193
BC00397=165709,388705,1075193
BC00398=165709,388705,1075193
BC00399=170177,393849,1075193
BC00400=167581,390589,1075193
BC00401=251336,357301,1075161
BC00402=285530,292059,1075139
BC00403=287197,286835,1075139
BC00404=266012,266073,1075139
BC00405=287864,284746,1075139
BC00406=287864,284746,1075139
BC00407=300310,286719,1075135
BC00408=287865,284746,1075136
BC00409=287865,284746,1075136
BC00410=287865,284746,1075136
BC00411=287865,284746,1075136
BC00412=287865,284746,1075136
BC00413=279306,291990,1075139
BC00414=279306,291990,1075139
BC00415=309148,355815,1075139
BC00416=309148,355815,1075139
BC00417=309148,355815,1075136
BC00418=309148,355815,1075139
BC00419=309148,355815,1075139
BC00420=309148,355815,1075136
BC00421=309148,355815,1075139
BC00422=309148,355815,1075139
BC00423=289264,317558,1075139
BC00424=145494,233235,1075139
BC00425=140837,229747,1075139
BC00426=140604,226760,1075139
BC00427=140605,226760,1075139
BC00428=140605,226760,1075139
BC00429=122537,236913,1075139
BC00430=131798,232630,1075136
BC00431=131798,232630,1075136
BC00432=84291,239513,1075139
BC00433=172642,235618,1075139
BC00434=170415,234251,1075139
BC00435=170415,234251,1075139
BC00436=170415,234251,1075139
BC00437=170415,234251,1075139
BC00438=164867,233321,1075139
BC00439=169989,236697,1075139
BC00440=105824,241109,1075139
BC00441=108282,235653,1075139
BC00442=109265,233471,1075136
BC00443=109265,233471,1075139
BC00444=109265,233471,1075139
BC00445=109265,233471,1075136
BC00446=103738,224976,1075139
BC00447=101586,230083,1075139
BC00448=180693,243652,1075139
BC00449=274713,263212,1075139
BC00450=330649,240203,1075139
BC00451=330649,240203,1075139
BC00452=331135,239089,1075139
BC00453=331135,239089,1075139
BC00454=331135,239089,1075139
BC00455=335838,239907,1075139
BC00456=381325,247767,1075137
BC00457=386029,248575,1075139
BC00458=386029,248575,1075139
BC00459=385543,249689,1075139
BC00460=385543,258980,1075139
BC00461=331396,370413,1075139
BC00462=331396,370413,1075139
BC00463=331396,370413,1075139
BC00464=331396,370413,1075139
BC00465=331396,370413,1075139
BC00466=331396,370413,1075139
BC00467=331396,370413,1075139
BC00468=331396,370413,1075138
BC00469=331396,370413,1075139
BC00470=331396,370413,1075139
BC00471=331396,370413,1075139
BC00472=331396,370413,1075139
BC00473=331396,370413,1075139
BC00474=331396,370413,1075139
BC00475=331396,370413,1075139
BC00476=331396,370413,1075138
BC00477=331396,370413,1075139
BC00478=331396,370413,1075139
BC00479=331396,340365,1075139
BC00480=331396,340365,1075139
BC00481=331396,340365,1075139
BC00482=331396,340365,1075139
BC00483=331396,340365,1075139
BC00484=331396,340365,1075139
BC00485=330649,514882,1075139
BC00486=154505,514882,1075139
BC00487=204883,514304,820550
BC00488=216477,460314,345947
BC00489=221056,438991,158507
BC00490=221983,434676,120575
BC00491=221983,434676,120575
BC00492=221983,434676,120575
BC00493=221983,434676,120575
BC00494=221983,434676,120575
BC00495=221983,434676,120575
BC00496=221983,434676,120575
BC00497=221983,434676,120575
BC00498=221983,434676,120575
BC00499=277830,435781,149366
BC00500=340580,438465,187892
BC00501=340580,438465,187892
BC00502=340580,438465,187892
BC00503=340580,438465,187892
BC00504=340580,438465,187892
BC00505=340580,438465,187892
BC00506=340580,438465,187892
BC00507=340713,465766,187001
BC00508=265051,465766,187001
BC00509=265051,465766,187001
BC00510=265051,465766,187001
BC00511=265051,465766,187001
BC00512=265051,465766,187001
BC00513=265051,465766,187001
BC00514=265051,465766,187001
BC00515=265051,465766,187001
BC00516=265051,465766,187001
BC00517=265051,465766,187001
BC00518=265051,465766,187001
BC00519=265051,465766,187001
BC00520=265051,465766,187001
BC00521=265051,465766,187001
BC00522=265051,465766,187001
BC00523=265051,465766,187001
BC00524=265051,465766,187001
BC00525=265051,465766,187001
BC00526=265051,465766,187001
BC00527=265051,465766,187001
BC00528=286147,481014,186503
BC00529=340979,520647,185210
BC00530=119021,520647,185210
BC00531=118360,390509,385345
BC00532=117845,368543,271032
BC00533=117845,368543,271032
BC00534=117845,368543,271032
BC00535=117845,368543,271032
BC00536=117845,368543,271032
BC00537=117845,368543,271032
BC00538=117845,368543,271032
BC00539=101209,360863,304275
BC00540=101209,360863,304275
BC00541=101209,360863,304275
BC00542=101209,360863,304275
BC00543=101209,360863,304275
BC00544=101209,360863,304275
BC00545=101209,360863,304275
BC00546=101209,360863,304275
BC00547=118360,390509,385345
BC00548=119021,520647,185210
BC00549=340979,520647,185210
BC00550=249445,427787,239249
BC00551=249445,427787,239249
BC00552=249445,427787,239249
BC00553=249445,427787,239249
BC00554=249445,427787,239249
BC00555=249445,427787,239249
BC00556=249445,427787,239249
BC00557=249445,427787,239249
BC00558=249446,427788,239248
BC00559=249445,427787,239249
BC00560=249445,427787,239249
BC00561=249445,427787,239249
BC00562=249445,427787,239249
BC00563=249445,427787,239249
BC00564=249445,427787,239249
BC00565=249445,427787,239249
BC00566=249445,427787,239249
BC00567=249445,427787,239249
BC00568=239702,439068,205328
BC00569=180729,507346,17
BC00570=180729,507346,17
BC00571=180729,507346,17
BC00572=180729,507346,17
BC00573=180729,507346,17
BC00574=180729,507346,17
BC00575=180729,507346,17
BC00576=180729,507346,17
BC00577=276406,484220,79871
BC00578=340979,520647,185210
BC00579=119021,520647,185210
BC00580=118360,390509,385345
BC00581=97843,363369,456609
BC00582=111700,357406,379613
BC00583=111700,357406,379613
BC00584=111700,357406,379613
BC00585=111700,357406,379613
BC00586=111700,357406,379613
BC00587=111700,357406,379613
BC00588=111700,357406,379613
BC00589=111700,357406,379613
BC00590=118360,390509,385345
BC00591=119021,508950,185210
BC00592=340979,507059,185210
BC00593=340979,507059,185210
BC00594=321821,455628,215045
BC00595=285116,420221,235586
BC00596=280467,416791,237575
BC00597=279224,416680,237640
BC00598=307285,416607,237682
BC00599=307285,416607,237682
BC00600=279224,416680,237640
BC00601=279224,416680,237640
BC00602=303364,450008,223981
BC00603=316300,467868,216662
BC00604=316300,467868,216662
BC00605=316300,467868,216662
BC00606=316300,467868,216662
BC00607=316300,467868,216662
BC00608=316300,467868,216662
BC00609=316300,467868,216662
BC00610=316300,467868,216662
BC00611=340979,512522,185210
BC00612=119021,514342,185210
BC00613=118360,390509,385345
BC00614=143975,361174,462326
BC00615=143975,361174,408559
BC00616=143975,361174,408559
BC00617=143975,361174,408559
BC00618=143975,361174,408559
BC00619=143975,361174,408559
BC00620=143975,361174,408559
BC00621=143975,361174,462326
BC00622=118360,390509,385345
BC00623=119021,520647,185210
BC00624=340979,520647,185210
BC00625=343718,468217,172125
BC00626=332917,431078,162856
BC00627=320175,431078,162856
BC00628=307432,431079,162855
BC00629=307433,431078,162856
BC00630=307433,431078,162856
BC00631=307432,431079,162855
BC00632=320175,431078,162856
BC00633=320175,431078,162856
BC00634=345358,462914,137681
BC00635=345358,462914,137681
BC00636=345358,462914,137681
BC00637=345358,462914,137681
BC00638=345358,462914,137681
BC00639=345358,462914,137681
BC00640=345358,462914,137681
BC00641=345358,462914,137681
BC00642=340309,396589,137906
BC00643=340309,396589,137906
BC00644=333293,396589,137906
BC00645=340309,396589,137906
BC00646=340309,396589,137906
BC00647=328784,396589,137906
BC00648=329025,396589,137906
BC00649=340309,396589,137906
BC00650=311573,406866,180953
BC00651=322964,407308,182805
BC00652=318645,407308,182805
BC00653=339313,407308,182805
BC00654=339313,407308,182805
BC00655=304194,407308,182805
BC00656=298765,405067,182805
BC00657=317970,406128,182805
BC00658=334834,430175,216666
BC00659=366690,430175,216666
BC00660=348044,430175,216666
BC00661=366690,430175,216666
BC00662=366690,430175,216666
BC00663=339780,430175,216666
BC00664=339083,427566,216666
BC00665=366690,430175,216666
EC00000=-798156,-1296783
EC00001=-798156,-1296783
EC00002=-798156,-1296783
EC00003=-798156,-1296783
EC00004=-798156,-1296783
EC00005=-798156,-1296783
EC00006=-798156,-1296783
EC00007=-798156,-1296783
EC00008=-798156,-1296783
EC00009=-798156,-1296783
EC00010=-798156,-1296783
EC00011=-798156,-1296783
EC00012=-798156,-1296783
EC00013=-798156,-1296783
EC00014=-798156,-1296783
EC00015=-798156,-1296783
EC00016=-798156,-1296783
EC00017=-798156,-1296783
EC00018=-798155,-1296782
EC00019=-798156,-1296783
EC00020=-798156,-1296783
EC00021=-798156,-1296783
EC00022=-798156,-1296783
EC00023=-798156,-1296783
EC00024=-798156,-1296783
EC00025=-798156,-1296783
EC00026=-798156,-1296783
EC00027=-798156,-1296783
EC00028=-798156,-1296783
EC00029=-798156,-1296783
EC00030=-798156,-1296783
EC00031=-798156,-1296783
EC00032=-798156,-1296783
EC00033=-798156,-1296783
EC00034=-798156,-1296783
EC00035=-798156,-1296783
EC00036=-798156,-1296783
EC00037=-798156,-1296783
EC00038=-798156,-1296783
EC00039=-798156,-1296783
EC00040=-798156,-1296783
EC00041=-798156,-1296783
EC00042=-798156,-1296783
EC00043=-798156,-1296783
EC00044=-798156,-1296783
EC00045=-798156,-1296783
EC00046=-798156,-1296783
EC00047=-798156,-1296783
EC00048=-798156,-1296783
EC00049=-798156,-1296783
EC00050=-798156,-1296783
EC00051=-975524,-1296783
EC00052=-975524,-1296783
EC00053=-975524,-1296783
EC00054=-975524,-1296783
EC00055=-975524,-1296783
EC00056=-975524,-1296783
EC00057=-975524,-1296783
EC00058=-975524,-1296783
EC00059=-975524,-1296783
EC00060=-975524,-1296783
EC00061=-975524,-1296783
EC00062=-975524,-1296783
EC00063=-975524,-1296783
EC00064=-975524,-1296783
EC00065=-975524,-1296783
EC00066=-975524,-1296783
EC00067=-975524,-1296783
EC00068=-975524,-1296783
EC00069=-975524,-1296783
EC00070=-975524,-1296783
EC00071=-975524,-1296783
EC00072=-975524,-1296783
EC00073=-975522,-1296782
EC00074=-975522,-1296782
EC00075=-975522,-1296782
EC00076=-975522,-1296782
EC00077=-975522,-1296782
EC00078=-975522,-1296782
EC00079=-975522,-1296782
EC00080=-975522,-1296782
EC00081=-975522,-1296782
EC00082=-975524,-1296783
EC00083=-975524,-1296783
EC00084=-879601,-1296783
EC00085=-798154,-1296782
EC00086=-798154,-1296782
EC00087=-798154,-1296782
EC00088=-798154,-1296782
EC00089=-798154,-1296782
EC00090=-798154,-1296782
EC00091=-798154,-1296782
EC00092=-798154,-1296782
EC00093=-798154,-1296782
EC00094=-798154,-1296782
EC00095=-798154,-1296782
EC00096=-798154,-1296782
EC00097=-798154,-1296782
EC00098=-798156,-1296783
EC00099=-798156,-1296783
EC00100=-798156,-1296783
EC00101=-798156,-1296783
EC00102=-798156,-1296783
EC00103=-798156,-1296783
EC00104=-798156,-1296783
EC00105=-798156,-1296783
EC00106=-798156,-1296783
EC00107=-798156,-1296783
EC00108=-798156,-1296783
EC00109=-798156,-1296783
EC00110=-798156,-1296783
EC00111=-798156,-1296783
EC00112=-798156,-1296783
EC00113=-798156,-1296783
EC00114=-798156,-1296783
EC00115=-798156,-1296783
EC00116=-798156,-1296783
EC00117=-798156,-1296783
EC00118=-798156,-1296783
EC00119=-798156,-1296783
EC00120=-798156,-1296783
EC00121=-798156,-1296783
EC00122=-798156,-1296783
EC00123=-798156,-1296783
EC00124=-798156,-1296783
EC00125=-798156,-1296783
EC00126=-798156,-1296783
EC00127=-798156,-1296783
EC00128=-798156,-1296783
EC00129=-798156,-1296783
EC00130=-798156,-1296783
EC00131=-798156,-1296783
EC00132=-798156,-1296783
EC00133=-798156,-1296783
EC00134=-798156,-1296783
EC00135=-798156,-1296783
EC00136=-798156,-1296783
EC00137=-798156,-1296783
EC00138=-798156,-1296783
EC00139=-798156,-1296783
EC00140=-798156,-1296783
EC00141=-798156,-1296783
EC00142=-798156,-1296783
EC00143=-798156,-1296783
EC00144=-798156,-1296783
EC00145=-798156,-1296783
EC00146=-798156,-1296783
EC00147=-798156,-1296783
EC00148=-798156,-1296783
EC00149=-798156,-1296783
EC00150=-798156,-1296783
EC00151=-798156,-1296783
EC00152=-798156,-1296783
EC00153=-798156,-1296783
EC00154=-798156,-1296783
EC00155=-798156,-1296783
EC00156=-798156,-1296783
EC00157=-798156,-1296783
EC00158=-798156,-1296783
EC00159=-798156,-1296783
EC00160=-798156,-1296783
EC00161=-798156,-1296783
EC00162=-798156,-1296783
EC00163=-798156,-1296783
EC00164=-798156,-1296783
EC00165=-798156,-1296783
EC00166=-798156,-1296783
EC00167=-798154,-1296781
EC00168=-798154,-1296781
EC00169=-798154,-1296781
EC00170=-798154,-1296781
EC00171=-798156,-1296783
EC00172=-798156,-1296783
EC00173=-798156,-1296783
EC00174=-798156,-1296783
EC00175=-798156,-1296783
EC00176=-798156,-1296783
EC00177=-798156,-1296783
EC00178=-798156,-1296783
EC00179=-798156,-1296783
EC00180=-798156,-1296783
EC00181=-798156,-1296783
EC00182=-798156,-1296783
EC00183=-798156,-1296783
EC00184=-798156,-1296783
EC00185=-798156,-1296783
EC00186=-798156,-1296783
EC00187=-798156,-1296783
EC00188=-798156,-1296783
EC00189=-798156,-1296783
EC00190=-798156,-1296783
EC00191=-798156,-1296783
EC00192=-798156,-1296783
EC00193=-798156,-1296783
EC00194=-798156,-1296783
EC00195=-798156,-1296783
EC00196=-798156,-1296783
EC00197=-798156,-1296783
EC00198=-798156,-1296783
EC00199=-798156,-1296783
EC00200=-798156,-1296783
EC00201=-798156,-1296783
EC00202=-798156,-1296783
EC00203=-798156,-1296783
EC00204=-798156,-1296783
EC00205=-798156,-1296783
EC00206=-798156,-1296783
EC00207=-798156,-1296783
EC00208=-798156,-1296783
EC00209=-798156,-1296783
EC00210=-798156,-1296783
EC00211=-798156,-1296783
EC00212=-798156,-1296783
EC00213=-798156,-1296783
EC00214=-798156,-1296783
EC00215=-798156,-1296783
EC00216=-798156,-1296783
EC00217=-798156,-1296783
EC00218=-798156,-1296783
EC00219=-798156,-1296783
EC00220=-798156,-1296783
EC00221=-798156,-1296783
EC00222=-798156,-1296783
EC00223=-798156,-1296783
EC00224=-798156,-1296783
EC00225=-798153,-1296779
EC00226=-798153,-1296779
EC00227=-798156,-1296783
EC00228=-798156,-1296783
EC00229=-798156,-1296783
EC00230=-798156,-1296783
EC00231=-798156,-1296783
EC00232=-798155,-1296781
EC00233=-798156,-1296783
EC00234=-798156,-1296783
EC00235=-798155,-1296781
EC00236=-798155,-1296781
EC00237=-798154,-1296780
EC00238=-798152,-1296778
EC00239=-798152,-1296778
EC00240=-798153,-1296779
EC00241=-875273,-1296783
EC00242=-975524,-1296783
EC00243=-975524,-1296783
EC00244=-975524,-1296783
EC00245=-975524,-1296783
EC00246=-975524,-1296783
EC00247=-975524,-1296783
EC00248=-975524,-1296783
EC00249=-975524,-1296783
EC00250=-975524,-1296783
EC00251=-975524,-1296783
EC00252=-975524,-1296783
EC00253=-975524,-1296783
EC00254=-975524,-1296783
EC00255=-975524,-1296783
EC00256=-975524,-1296783
EC00257=-975524,-1296783
EC00258=-975524,-1296783
EC00259=-975524,-1296783
EC00260=-975524,-1296783
EC00261=-975524,-1296783
EC00262=-975524,-1296783
EC00263=-975524,-1296783
EC00264=-975524,-1296783
EC00265=-975524,-1296783
EC00266=-975518,-1296781
EC00267=-975518,-1296781
EC00268=-975524,-1296783
EC00269=-975524,-1296783
EC00270=-975524,-1296783
EC00271=-798156,-1296783
EC00272=-798156,-1296783
EC00273=-798156,-1296783
EC00274=-975524,-1296783
EC00275=-975524,-1296783
EC00276=-798156,-1296783
EC00277=-798156,-1296783
EC00278=-798156,-1296783
EC00279=-798156,-1296783
EC00280=-798156,-1296783
EC00281=-798156,-1296783
EC00282=-798156,-1296783
EC00283=-798156,-1296783
EC00284=-798156,-1296783
EC00285=-975524,-1296783
EC00286=-975524,-1296783
EC00287=-798156,-1296783
EC00288=-798156,-1296783
EC00289=-798156,-1296783
EC00290=-798156,-1296783
EC00291=-798156,-1296783
EC00292=-798156,-1296783
EC00293=-798156,-1296783
EC00294=-798156,-1296783
EC00295=-798156,-1296783
EC00296=-798156,-1296783
EC00297=-798156,-1296783
EC00298=-798156,-1296783
EC00299=-798156,-1296783
EC00300=-798156,-1296783
EC00301=-798156,-1296783
EC00302=-798156,-1296783
EC00303=-798156,-1296783
EC00304=-798156,-1296783
EC00305=-798156,-1296783
EC00306=-798154,-1296780
EC00307=-798154,-1296782
EC00308=-798154,-1296782
EC00309=-798154,-1296782
EC00310=-798156,-1296783
EC00311=-798156,-1296783
EC00312=-798156,-1296783
EC00313=-798156,-1296783
EC00314=-798156,-1296783
EC00315=-798156,-1296783
EC00316=-798156,-1296783
EC00317=-798156,-1296783
EC00318=-798156,-1296783
EC00319=-798156,-1296783
EC00320=-798156,-1296783
EC00321=-798156,-1296783
EC00322=-798156,-1296783
EC00323=-798156,-1296783
EC00324=-798154,-1296781
EC00325=-798154,-1296781
EC00326=-798154,-1296781
EC00327=-798154,-1296781
EC00328=-798154,-1296781
EC00329=-798154,-1296783
EC00330=-798156,-1296783
EC00331=-798156,-1296783
EC00332=-798156,-1296783
EC00333=-798154,-1296782
EC00334=-798156,-1296783
EC00335=-798156,-1296783
EC00336=-798156,-1296783
EC00337=-798156,-1296783
EC00338=-798156,-1296783
EC00339=-798156,-1296783
EC00340=-798156,-1296783
EC00341=-798156,-1296783
EC00342=-798156,-1296783
EC00343=-798156,-1296783
EC00344=-798156,-1296783
EC00345=-798156,-1296783
EC00346=-798156,-1296783
EC00347=-798156,-1296783
EC00348=-798156,-1296783
EC00349=-798156,-1296783
EC00350=-798156,-1296783
EC00351=-798156,-1296783
EC00352=-798156,-1296783
EC00353=-798156,-1296783
EC00354=-798156,-1296783
EC00355=-798156,-1296783
EC00356=-798156,-1296783
EC00357=-798156,-1296783
EC00358=-798156,-1296783
EC00359=-798156,-1296783
EC00360=-798156,-1296783
EC00361=-798156,-1296783
EC00362=-798156,-1296783
EC00363=-798156,-1296783
EC00364=-798156,-1296783
EC00365=-798156,-1296783
EC00366=-798156,-1296783
EC00367=-798155,-1296782
EC00368=-798156,-1296783
EC00369=-798156,-1296783
EC00370=-798156,-1296783
EC00371=-798156,-1296783
EC00372=-898210,-1296783
EC00373=-975524,-1296783
EC00374=-975524,-1296783
EC00375=-975522,-1296782
EC00376=-975524,-1296783
EC00377=-975524,-1296783
EC00378=-975522,-1296782
EC00379=-975522,-1296782
EC00380=-975522,-1296782
EC00381=-975524,-1296783
EC00382=-975524,-1296783
EC00383=-975524,-1296783
EC00384=-975524,-1296783
EC00385=-975524,-1296783
EC00386=-975524,-1296783
EC00387=-975524,-1296783
EC00388=-975524,-1296783
EC00389=-975524,-1296783
EC00390=-975524,-1296783
EC00391=-975524,-1296783
EC00392=-975524,-1296783
EC00393=-975524,-1296783
EC00394=-975524,-1296783
EC00395=-975524,-1296783
EC00396=-975524,-1296783
EC00397=-975524,-1296783
EC00398=-975524,-1296783
EC00399=-975524,-1296783
EC00400=-975524,-1296783
EC00401=-868649,-1296783
EC00402=-798156,-1296783
EC00403=-798156,-1296783
EC00404=-798156,-1296783
EC00405=-798156,-1296783
EC00406=-798156,-1296783
EC00407=-798155,-1296781
EC00408=-798155,-1296782
EC00409=-798155,-1296782
EC00410=-798155,-1296782
EC00411=-798155,-1296782
EC00412=-798155,-1296782
EC00413=-798156,-1296783
EC00414=-798156,-1296783
EC00415=-798156,-1296783
EC00416=-798156,-1296783
EC00417=-798154,-1296781
EC00418=-798156,-1296783
EC00419=-798156,-1296783
EC00420=-798154,-1296781
EC00421=-798156,-1296783
EC00422=-798156,-1296783
EC00423=-798156,-1296783
EC00424=-798156,-1296783
EC00425=-798156,-1296783
EC00426=-798156,-1296783
EC00427=-798156,-1296783
EC00428=-798156,-1296783
EC00429=-798156,-1296783
EC00430=-798155,-1296782
EC00431=-798155,-1296782
EC00432=-798156,-1296783
EC00433=-798156,-1296783
EC00434=-798156,-1296783
EC00435=-798156,-1296783
EC00436=-798156,-1296783
EC00437=-798156,-1296783
EC00438=-798156,-1296783
EC00439=-798156,-1296783
EC00440=-798156,-1296783
EC00441=-798156,-1296783
EC00442=-798154,-1296782
EC00443=-798156,-1296783
EC00444=-798156,-1296783
EC00445=-798154,-1296782
EC00446=-798156,-1296783
EC00447=-798156,-1296783
EC00448=-798156,-1296783
EC00449=-798156,-1296783
EC00450=-798156,-1296783
EC00451=-798156,-1296783
EC00452=-798156,-1296783
EC00453=-798156,-1296783
EC00454=-798156,-1296783
EC00455=-798156,-1296783
EC00456=-798155,-1296782
EC00457=-798156,-1296783
EC00458=-798156,-1296783
EC00459=-798156,-1296783
EC00460=-798156,-1296783
EC00461=-798156,-1296783
EC00462=-798156,-1296783
EC00463=-798156,-1296783
EC00464=-798156,-1296783
EC00465=-798156,-1296783
EC00466=-798156,-1296783
EC00467=-798156,-1296783
EC00468=-798155,-1296781
EC00469=-798156,-1296783
EC00470=-798156,-1296783
EC00471=-798156,-1296783
EC00472=-798156,-1296783
EC00473=-798156,-1296783
EC00474=-798156,-1296783
EC00475=-798156,-1296783
EC00476=-798154,-1296782
EC00477=-798156,-1296783
EC00478=-798156,-1296783
EC00479=-798156,-1296783
EC00480=-798156,-1296783
EC00481=-798156,-1296783
EC00482=-798156,-1296783
EC00483=-798156,-1296783
EC00484=-798156,-1296783
EC00485=-798156,-1296783
EC00486=-798156,-1296783
EC00487=-798156,-1296783
EC00488=-798156,-1296783
EC00489=-798156,-1296783
EC00490=-798156,-1296783
EC00491=-798156,-1296783
EC00492=-798156,-1296783
EC00493=-798156,-1296783
EC00494=-798156,-1296783
EC00495=-798156,-1296783
EC00496=-798156,-1296783
EC00497=-798156,-1296783
EC00498=-798156,-1296783
EC00499=-798156,-1296783
EC00500=-798156,-1296783
EC00501=-798156,-1296783
EC00502=-798156,-1296783
EC00503=-798156,-1296783
EC00504=-798156,-1296783
EC00505=-798156,-1296783
EC00506=-798156,-1296783
EC00507=-798156,-1296783
EC00508=-798156,-1296783
EC00509=-798156,-1296783
EC00510=-798156,-1296783
EC00511=-798156,-1296783
EC00512=-798156,-1296783
EC00513=-798156,-1296783
EC00514=-798156,-1296783
EC00515=-798156,-1296783
EC00516=-798156,-1296783
EC00517=-798156,-1296783
EC00518=-798156,-1296783
EC00519=-798156,-1296783
EC00520=-798156,-1296783
EC00521=-798156,-1296783
EC00522=-798156,-1296783
EC00523=-798156,-1296783
EC00524=-798156,-1296783
EC00525=-798156,-1296783
EC00526=-798156,-1296783
EC00527=-798156,-1296783
EC00528=-798156,-1296783
EC00529=-798156,-1296783
EC00530=-798156,-1296783
EC00531=-798156,-1296783
EC00532=-798156,-1296783
EC00533=-798156,-1296783
EC00534=-798156,-1296783
EC00535=-798156,-1296783
EC00536=-798156,-1296783
EC00537=-798156,-1296783
EC00538=-798156,-1296783
EC00539=-798156,-1296783
EC00540=-798156,-1296783
EC00541=-798156,-1296783
EC00542=-798156,-1296783
EC00543=-798156,-1296783
EC00544=-798156,-1296783
EC00545=-798156,-1296783
EC00546=-798156,-1296783
EC00547=-798156,-1296783
EC00548=-798156,-1296783
EC00549=-798156,-1296783
EC00550=-798156,-1296783
EC00551=-798156,-1296783
EC00552=-798156,-1296783
EC00553=-798156,-1296783
EC00554=-798156,-1296783
EC00555=-798156,-1296783
EC00556=-798156,-1296783
EC00557=-798156,-1296783
EC00558=-798155,-1296782
EC00559=-798156,-1296783
EC00560=-798156,-1296783
EC00561=-798156,-1296783
EC00562=-798156,-1296783
EC00563=-798156,-1296783
EC00564=-798156,-1296783
EC00565=-798156,-1296783
EC00566=-798156,-1296783
EC00567=-798156,-1296783
EC00568=-798156,-1296783
EC00569=-798156,-1296783
EC00570=-798156,-1296783
EC00571=-798156,-1296783
EC00572=-798156,-1296783
EC00573=-798156,-1296783
EC00574=-798156,-1296783
EC00575=-798156,-1296783
EC00576=-798156,-1296783
EC00577=-798156,-1296783
EC00578=-798156,-1296783
EC00579=-798156,-1296783
EC00580=-798156,-1296783
EC00581=-798156,-1296783
EC00582=-798156,-1296783
EC00583=-798156,-1296783
EC00584=-798156,-1296783
EC00585=-798156,-1296783
EC00586=-798156,-1296783
EC00587=-798156,-1296783
EC00588=-798156,-1296783
EC00589=-798156,-1296783
EC00590=-798156,-1296783
EC00591=-798156,-1296783
EC00592=-798156,-1296783
EC00593=-798156,-1296783
EC00594=-798156,-1296783
EC00595=-798156,-1296783
EC00596=-798156,-1296783
EC00597=-798156,-1296783
EC00598=-798156,-1296783
EC00599=-798156,-1296783
EC00600=-798156,-1296783
EC00601=-798156,-1296783
EC00602=-798156,-1296783
EC00603=-798156,-1296783
EC00604=-798156,-1296783
EC00605=-798156,-1296783
EC00606=-798156,-1296783
EC00607=-798156,-1296783
EC00608=-798156,-1296783
EC00609=-798156,-1296783
EC00610=-798156,-1296783
EC00611=-798156,-1296783
EC00612=-798156,-1296783
EC00613=-798156,-1296783
EC00614=-798156,-1296783
EC00615=-798156,-1296783
EC00616=-798156,-1296783
EC00617=-798156,-1296783
EC00618=-798156,-1296783
EC00619=-798156,-1296783
EC00620=-798156,-1296783
EC00621=-798156,-1296783
EC00622=-798156,-1296783
EC00623=-798156,-1296783
EC00624=-798156,-1296783
EC00625=-798156,-1296783
EC00626=-798156,-1296783
EC00627=-798156,-1296783
EC00628=-798155,-1296782
EC00629=-798156,-1296783
EC00630=-798156,-1296783
EC00631=-798155,-1296782
EC00632=-798156,-1296783
EC00633=-798156,-1296783
EC00634=-798156,-1296783
EC00635=-798156,-1296783
EC00636=-798156,-1296783
EC00637=-798156,-1296783
EC00638=-798156,-1296783
EC00639=-798156,-1296783
EC00640=-798156,-1296783
EC00641=-798156,-1296783
EC00642=-798156,-1296783
EC00643=-798156,-1296783
EC00644=-798156,-1296783
EC00645=-798156,-1296783
EC00646=-798156,-1296783
EC00647=-798156,-1296783
EC00648=-798156,-1296783
EC00649=-798156,-1296783
EC00650=-798156,-1296783
EC00651=-798156,-1296783
EC00652=-798156,-1296783
EC00653=-798156,-1296783
EC00654=-798156,-1296783
EC00655=-798156,-1296783
EC00656=-798156,-1296783
EC00657=-798156,-1296783
EC00658=-798156,-1296783
EC00659=-798156,-1296783
EC00660=-798156,-1296783
EC00661=-798156,-1296783
EC00662=-798156,-1296783
EC00663=-798156,-1296783
EC00664=-798156,-1296783
EC00665=-798156,-1296783
///POSTYPE BASE
///RECTAN
///RCONF 0,0,0,0,1,0,0,0,0,0,0,0,0,0,0,0,0,0,0,0,0,0,0,0
P00006=2.006,1.622,-0.565,0.0000,0.0000,0.0000
P00021=0.073,2.058,-0.109,0.0000,0.0000,0.0000
P00022=2.006,1.622,-0.565,0.0000,0.0000,0.0000
///RCONF 0,0,0,0,0,0,0,0,0,0,0,0,0,0,0,0,0,0,0,0,0,0,0,0
P00023=-2.957,-4.083,2.762,0.0000,0.0000,0.0000
P00031=-0.170,0.039,-0.647,0.0000,0.0000,0.0000
P00032=-0.423,0.157,3.222,0.0000,0.0000,0.0000
P00033=0.854,-1.099,3.047,0.0000,0.0000,0.0000
///RCONF 0,0,0,0,1,0,0,0,0,0,0,0,0,0,0,0,0,0,0,0,0,0,0,0
P00034=-8.151,9.743,-4.393,0.0000,0.0000,0.0000
///RCONF 0,0,0,0,0,0,0,0,0,0,0,0,0,0,0,0,0,0,0,0,0,0,0,0
P00035=0.390,-0.027,1.040,0.0000,0.0000,0.0000
P00036=-2.434,0.084,0.197,0.0000,0.0000,0.0000
P00037=-1.075,5.090,-3.949,0.0000,0.0000,0.0000
P00038=0.174,-1.527,-10.860,0.0000,0.0000,0.0000
P00039=-0.109,1.838,-0.266,0.0000,0.0000,0.0000
P00040=2.716,-0.016,3.014,0.0000,0.0000,0.0000
P00041=-0.109,0.014,0.966,0.0000,0.0000,0.0000
P00042=-0.220,0.371,-0.613,0.0000,0.0000,0.0000
P00043=-0.179,-5.890,-3.227,0.0000,0.0000,0.0000
P00051=-5.945,4.696,-10.293,0.0000,0.0000,0.0000
P00052=-0.153,5.586,-7.982,0.0000,0.0000,0.0000
P00055=-0.009,2.790,-4.790,0.0000,0.0000,0.0000
P00056=3.147,0.012,0.038,0.0000,0.0000,0.0000
P00057=13.307,-11.525,-2.645,0.0000,0.0000,0.0000
P00058=6.894,-13.094,-1.754,0.0000,0.0000,0.0000
P00059=-2.448,-6.714,-12.718,0.0000,0.0000,0.0000
P00060=1524.284,698.404,-261.973,-0.4635,36.8346,-1.2388
P00061=1211.499,975.999,-261.374,0.5148,35.2356,175.5099
P00090=-14.057,13.261,-6.464,0.0000,0.0000,0.0000
P00091=1.048,0.648,3.624,0.0000,0.0000,0.0000
//INST
///DATE 2024/11/25 14:59
///ATTR SC,RW
///GROUP1 RB1,BS1
///GROUP2 ST1
NOP
'OK_r2_O8B-O21B(90,0)
'Path S3645
SFTOF3D
'POW POP KM
MOVJ C00000 BC00000 VJ=100.00  +MOVJ EC00000 VJ=100.00
MOVL C00001 BC00001 V=666.7  +MOVJ EC00001 VJ=100.00
SMOVL C00002 BC00002 V=166.7  +MOVJ EC00002
SREFP 3 C00003 BC00003  +REFP EC00003
CALL JOB:SEARCH-R1-S13D
SET P031 P006
SFTON3D P031
SMOVL C00004 BC00004 V=166.7  +MOVJ EC00004
SREFP 3 C00005 BC00005  +REFP EC00005
CALL JOB:SEARCH-R1-S13D
SET P031 P006
SFTON3D P031
SFTOF3D
SMOVL C00006 BC00006 V=166.7  +MOVJ EC00006
MOVL C00007 BC00007 V=666.7  +MOVJ EC00007 VJ=100.00
SMOVL C00008 BC00008 V=166.7  +MOVJ EC00008
SREFP 3 C00009 BC00009  +REFP EC00009
CALL JOB:SEARCH-R1-S13D
SET P051 P006
SFTON3D P051
SMOVL C00010 BC00010 V=166.7  +MOVJ EC00010
SREFP 3 C00011 BC00011  +REFP EC00011
CALL JOB:SEARCH-R1-S13D
SET P051 P006
SFTON3D P051
SMOVL C00012 BC00012 V=166.7  +MOVJ EC00012
MOVL C00013 BC00013 V=1000.0  +MOVJ EC00013 VJ=100.00
'Path S3646
SFTOF3D
MOVJ C00014 BC00014 VJ=100.00  +MOVJ EC00014 VJ=100.00
MOVL C00015 BC00015 V=666.7  +MOVJ EC00015 VJ=100.00
SMOVL C00016 BC00016 V=333.3  +MOVJ EC00016
SMOVL C00017 BC00017 V=166.7  +MOVJ EC00017
SREFP 3 C00018 BC00018  +REFP EC00018
CALL JOB:SEARCH-R1-S13D
SET P035 P006
SFTON3D P035
SMOVL C00019 BC00019 V=166.7  +MOVJ EC00019
SMOVL C00020 BC00020 V=250.0  +MOVJ EC00020
SMOVL C00021 BC00021 V=166.7  +MOVJ EC00021
SREFP 3 C00022 BC00022  +REFP EC00022
CALL JOB:SEARCH-R1-S13D
SET P035 P006
SFTON3D P035
SMOVL C00023 BC00023 V=166.7  +MOVJ EC00023
SMOVL C00024 BC00024 V=166.7  +MOVJ EC00024
MOVL C00025 BC00025 V=666.7  +MOVJ EC00025 VJ=100.00
MOVL C00026 BC00026 V=1000.0  +MOVJ EC00026 VJ=100.00
MOVJ C00027 BC00027 VJ=100.00  +MOVJ EC00027 VJ=100.00
'Path S3647
SFTOF3D
MOVJ C00028 BC00028 VJ=100.00  +MOVJ EC00028 VJ=100.00
MOVJ C00029 BC00029 VJ=100.00  +MOVJ EC00029 VJ=100.00
MOVL C00030 BC00030 V=666.7  +MOVJ EC00030 VJ=100.00
SMOVL C00031 BC00031 V=166.7  +MOVJ EC00031
SREFP 3 C00032 BC00032  +REFP EC00032
CALL JOB:SEARCH-R1-S13D
SET P032 P006
SFTON3D P032
SMOVL C00033 BC00033 V=166.7  +MOVJ EC00033
SREFP 3 C00034 BC00034  +REFP EC00034
CALL JOB:SEARCH-R1-S13D
SET P032 P006
SFTON3D P032
SMOVL C00035 BC00035 V=166.7  +MOVJ EC00035
SREFP 3 C00036 BC00036  +REFP EC00036
CALL JOB:SEARCH-R1-S13D
SET P032 P006
SFTON3D P032
SMOVL C00037 BC00037 V=166.7  +MOVJ EC00037
MOVL C00038 BC00038 V=666.7  +MOVJ EC00038 VJ=100.00
MOVL C00039 BC00039 V=1000.0  +MOVJ EC00039 VJ=100.00
'Path S3648
SFTOF3D
MOVJ C00040 BC00040 VJ=100.00  +MOVJ EC00040 VJ=100.00
MOVL C00041 BC00041 V=666.7  +MOVJ EC00041 VJ=100.00
SMOVL C00042 BC00042 V=166.7  +MOVJ EC00042
SREFP 3 C00043 BC00043  +REFP EC00043
CALL JOB:SEARCH-R1-S13D
SET P033 P006
SFTON3D P033
SMOVL C00044 BC00044 V=166.7  +MOVJ EC00044
SREFP 3 C00045 BC00045  +REFP EC00045
CALL JOB:SEARCH-R1-S13D
SET P033 P006
SFTON3D P033
SMOVL C00046 BC00046 V=166.7  +MOVJ EC00046
SMOVL C00047 BC00047 V=250.0  +MOVJ EC00047
SMOVL C00048 BC00048 V=166.7  +MOVJ EC00048
SREFP 3 C00049 BC00049  +REFP EC00049
CALL JOB:SEARCH-R1-S13D
SET P033 P006
SFTON3D P033
SMOVL C00050 BC00050 V=166.7  +MOVJ EC00050
MOVL C00051 BC00051 V=1000.0  +MOVJ EC00051 VJ=100.00
MOVJ C00052 BC00052 VJ=100.00  +MOVJ EC00052 VJ=100.00
'Path S3649
SFTOF3D
MOVJ C00053 BC00053 VJ=100.00  +MOVJ EC00053 VJ=100.00
MOVL C00054 BC00054 V=666.7  +MOVJ EC00054 VJ=100.00
SMOVL C00055 BC00055 V=166.7  +MOVJ EC00055
SREFP 3 C00056 BC00056  +REFP EC00056
CALL JOB:SEARCH-R1-S13D
SET P038 P006
SFTON3D P038
SMOVL C00057 BC00057 V=166.7  +MOVJ EC00057
SMOVL C00058 BC00058 V=250.0  +MOVJ EC00058
SMOVL C00059 BC00059 V=166.7  +MOVJ EC00059
SREFP 3 C00060 BC00060  +REFP EC00060
CALL JOB:SEARCH-R1-S13D
SET P038 P006
SFTON3D P038
SMOVL C00061 BC00061 V=166.7  +MOVJ EC00061
SMOVL C00062 BC00062 V=166.7  +MOVJ EC00062
SMOVL C00063 BC00063 V=166.7  +MOVJ EC00063
SREFP 3 C00064 BC00064  +REFP EC00064
CALL JOB:SEARCH-R1-S13D
SET P038 P006
SFTON3D P038
SMOVL C00065 BC00065 V=166.7  +MOVJ EC00065
SMOVL C00066 BC00066 V=200.0  +MOVJ EC00066
SMOVL C00067 BC00067 V=250.0  +MOVJ EC00067
MOVL C00068 BC00068 V=666.7  +MOVJ EC00068 VJ=100.00
MOVL C00069 BC00069 V=1000.0  +MOVJ EC00069 VJ=100.00
MOVJ C00070 BC00070 VJ=100.00  +MOVJ EC00070 VJ=100.00
'Path S3650
SFTOF3D
MOVJ C00071 BC00071 VJ=100.00  +MOVJ EC00071 VJ=100.00
MOVL C00072 BC00072 V=666.7  +MOVJ EC00072 VJ=100.00
SMOVL C00073 BC00073 V=166.7  +MOVJ EC00073
SREFP 3 C00074 BC00074  +REFP EC00074
CALL JOB:SEARCH-R1-S13D
SET P040 P006
SFTON3D P040
SMOVL C00075 BC00075 V=166.7  +MOVJ EC00075
SREFP 3 C00076 BC00076  +REFP EC00076
CALL JOB:SEARCH-R1-S13D
SET P040 P006
SFTON3D P040
SMOVL C00077 BC00077 V=166.7  +MOVJ EC00077
SMOVL C00078 BC00078 V=250.0  +MOVJ EC00078
SMOVL C00079 BC00079 V=166.7  +MOVJ EC00079
SREFP 3 C00080 BC00080  +REFP EC00080
CALL JOB:SEARCH-R1-S13D
SET P040 P006
SFTON3D P040
SMOVL C00081 BC00081 V=166.7  +MOVJ EC00081
MOVL C00082 BC00082 V=666.7  +MOVJ EC00082 VJ=100.00
MOVL C00083 BC00083 V=1000.0  +MOVJ EC00083 VJ=100.00
MOVJ C00084 BC00084 VJ=100.00  +MOVJ EC00084 VJ=100.00
'Path S3651
SFTOF3D
MOVJ C00085 BC00085 VJ=100.00  +MOVJ EC00085 VJ=100.00
MOVL C00086 BC00086 V=666.7  +MOVJ EC00086 VJ=100.00
SMOVL C00087 BC00087 V=166.7  +MOVJ EC00087
SREFP 3 C00088 BC00088  +REFP EC00088
CALL JOB:SEARCH-R1-S13D
SET P036 P006
SFTON3D P036
SMOVL C00089 BC00089 V=166.7  +MOVJ EC00089
SREFP 3 C00090 BC00090  +REFP EC00090
CALL JOB:SEARCH-R1-S13D
SET P036 P006
SFTON3D P036
SMOVL C00091 BC00091 V=166.7  +MOVJ EC00091
MOVJ C00092 BC00092 VJ=100.00  +MOVJ EC00092 VJ=100.00
MOVJ C00093 BC00093 VJ=100.00  +MOVJ EC00093 VJ=50.00
SMOVL C00094 BC00094 V=166.7  +MOVJ EC00094
SREFP 3 C00095 BC00095  +REFP EC00095
CALL JOB:SEARCH-R1-S13D
SET P036 P006
SFTON3D P036
SMOVL C00096 BC00096 V=166.7  +MOVJ EC00096
MOVL C00097 BC00097 V=666.7  +MOVJ EC00097 VJ=100.00
MOVJ C00098 BC00098 VJ=100.00  +MOVJ EC00098 VJ=100.00
'Path S3652
SFTOF3D
MOVJ C00099 BC00099 VJ=100.00  +MOVJ EC00099 VJ=100.00
MOVL C00100 BC00100 V=666.7  +MOVJ EC00100 VJ=100.00
SMOVL C00101 BC00101 V=166.7  +MOVJ EC00101
SREFP 3 C00102 BC00102  +REFP EC00102
CALL JOB:SEARCH-R1-S13D
SET P037 P006
SFTON3D P037
SMOVL C00103 BC00103 V=166.7  +MOVJ EC00103
SREFP 3 C00104 BC00104  +REFP EC00104
CALL JOB:SEARCH-R1-S13D
SET P037 P006
SFTON3D P037
SMOVL C00105 BC00105 V=166.7  +MOVJ EC00105
MOVL C00106 BC00106 V=666.7  +MOVJ EC00106 VJ=100.00
MOVL C00107 BC00107 V=1000.0  +MOVJ EC00107 VJ=100.00
'Path S3653
SFTOF3D
MOVJ C00108 BC00108 VJ=100.00  +MOVJ EC00108 VJ=100.00
MOVL C00109 BC00109 V=666.7  +MOVJ EC00109 VJ=100.00
SMOVL C00110 BC00110 V=166.7  +MOVJ EC00110
SREFP 3 C00111 BC00111  +REFP EC00111
CALL JOB:SEARCH-R1-S13D
SET P041 P006
SFTON3D P041
SMOVL C00112 BC00112 V=166.7  +MOVJ EC00112
SREFP 3 C00113 BC00113  +REFP EC00113
CALL JOB:SEARCH-R1-S13D
SET P041 P006
SFTON3D P041
SFTOF3D
SMOVL C00114 BC00114 V=166.7  +MOVJ EC00114
SMOVL C00115 BC00115 V=666.7  +MOVJ EC00115
SMOVL C00116 BC00116 V=166.7  +MOVJ EC00116
SREFP 3 C00117 BC00117  +REFP EC00117
CALL JOB:SEARCH-R1-S13D
SET P052 P006
SFTON3D P052
SMOVL C00118 BC00118 V=166.7  +MOVJ EC00118
SREFP 3 C00119 BC00119  +REFP EC00119
CALL JOB:SEARCH-R1-S13D
SET P052 P006
SFTON3D P052
SMOVL C00120 BC00120 V=166.7  +MOVJ EC00120
MOVL C00121 BC00121 V=1000.0  +MOVJ EC00121 VJ=100.00
'Path S3654
SFTOF3D
MOVJ C00122 BC00122 VJ=100.00  +MOVJ EC00122 VJ=100.00
MOVL C00123 BC00123 V=666.7  +MOVJ EC00123 VJ=100.00
SMOVL C00124 BC00124 V=166.7  +MOVJ EC00124
SREFP 3 C00125 BC00125  +REFP EC00125
CALL JOB:SEARCH-R1-S13D
SET P042 P006
SFTON3D P042
SMOVL C00126 BC00126 V=250.0  +MOVJ EC00126
SMOVL C00127 BC00127 V=166.7  +MOVJ EC00127
SREFP 3 C00128 BC00128  +REFP EC00128
CALL JOB:SEARCH-R1-S13D
SET P042 P006
SFTON3D P042
SMOVL C00129 BC00129 V=250.0  +MOVJ EC00129
MOVL C00130 BC00130 V=666.7  +MOVJ EC00130 VJ=100.00
MOVL C00131 BC00131 V=1000.0  +MOVJ EC00131 VJ=100.00
MOVJ C00132 BC00132 VJ=100.00  +MOVJ EC00132 VJ=100.00
'Path S3655
SFTOF3D
MOVJ C00133 BC00133 VJ=100.00  +MOVJ EC00133 VJ=100.00
MOVL C00134 BC00134 V=666.7  +MOVJ EC00134 VJ=100.00
SMOVL C00135 BC00135 V=166.7  +MOVJ EC00135
SREFP 3 C00136 BC00136  +REFP EC00136
CALL JOB:SEARCH-R1-S13D
SET P043 P006
SFTON3D P043
SMOVL C00137 BC00137 V=166.7  +MOVJ EC00137
SREFP 3 C00138 BC00138  +REFP EC00138
CALL JOB:SEARCH-R1-S13D
SET P043 P006
SFTON3D P043
SMOVL C00139 BC00139 V=166.7  +MOVJ EC00139
SMOVL C00140 BC00140 V=333.3  +MOVJ EC00140
SMOVL C00141 BC00141 V=166.7  +MOVJ EC00141
SREFP 3 C00142 BC00142  +REFP EC00142
CALL JOB:SEARCH-R1-S13D
SET P043 P006
SFTON3D P043
SFTOF3D
SMOVL C00143 BC00143 V=250.0  +MOVJ EC00143
MOVL C00144 BC00144 V=666.7  +MOVJ EC00144 VJ=100.00
MOVL C00145 BC00145 V=1000.0  +MOVJ EC00145 VJ=100.00
SMOVL C00146 BC00146 V=666.7  +MOVJ EC00146
SMOVL C00147 BC00147 V=166.7  +MOVJ EC00147
SREFP 3 C00148 BC00148  +REFP EC00148
CALL JOB:SEARCH-R1-S13D
SET P055 P006
SFTON3D P055
SMOVL C00149 BC00149 V=166.7  +MOVJ EC00149
SREFP 3 C00150 BC00150  +REFP EC00150
CALL JOB:SEARCH-R1-S13D
SET P055 P006
SFTON3D P055
SFTOF3D
SMOVL C00151 BC00151 V=166.7  +MOVJ EC00151
MOVJ C00152 BC00152 VJ=100.00  +MOVJ EC00152 VJ=100.00
MOVJ C00153 BC00153 VJ=100.00  +MOVJ EC00153 VJ=100.00
SMOVL C00154 BC00154 V=166.7  +MOVJ EC00154
SREFP 3 C00155 BC00155  +REFP EC00155
CALL JOB:SEARCH-R1-S13D
SET P056 P006
SFTON3D P056
SMOVL C00156 BC00156 V=166.7  +MOVJ EC00156
SREFP 3 C00157 BC00157  +REFP EC00157
CALL JOB:SEARCH-R1-S13D
SET P056 P006
SFTON3D P056
SMOVL C00158 BC00158 V=166.7  +MOVJ EC00158
MOVL C00159 BC00159 V=1000.0  +MOVJ EC00159 VJ=100.00
'Path S3656
SFTOF3D
MOVJ C00160 BC00160 VJ=100.00  +MOVJ EC00160 VJ=100.00
MOVL C00161 BC00161 V=666.7  +MOVJ EC00161 VJ=100.00
SMOVL C00162 BC00162 V=166.7  +MOVJ EC00162
SREFP 3 C00163 BC00163  +REFP EC00163
CALL JOB:SEARCH-R1-S13D
SET P039 P006
SFTON3D P039
SMOVL C00164 BC00164 V=166.7  +MOVJ EC00164
SREFP 3 C00165 BC00165  +REFP EC00165
CALL JOB:SEARCH-R1-S13D
SET P039 P006
SFTON3D P039
SMOVL C00166 BC00166 V=166.7  +MOVJ EC00166
SMOVL C00167 BC00167 V=333.3  +MOVJ EC00167
SMOVL C00168 BC00168 V=166.7  +MOVJ EC00168
SREFP 3 C00169 BC00169  +REFP EC00169
CALL JOB:SEARCH-R1-S13D
SET P039 P006
SFTON3D P039
SMOVL C00170 BC00170 V=166.7  +MOVJ EC00170
SMOVL C00171 BC00171 V=250.0  +MOVJ EC00171
SMOVL C00172 BC00172 V=416.7  +MOVJ EC00172
MOVL C00173 BC00173 V=666.7  +MOVJ EC00173 VJ=100.00
MOVL C00174 BC00174 V=1000.0  +MOVJ EC00174 VJ=100.00
'Path S3657
SFTOF3D
MOVJ C00175 BC00175 VJ=100.00  +MOVJ EC00175 VJ=100.00
MOVL C00176 BC00176 V=666.7  +MOVJ EC00176 VJ=100.00
SMOVL C00177 BC00177 V=166.7  +MOVJ EC00177
SREFP 3 C00178 BC00178  +REFP EC00178
CALL JOB:SEARCH-R1-S13D
SET P034 P006
SFTON3D P034
SMOVL C00179 BC00179 V=166.7  +MOVJ EC00179
SMOVL C00180 BC00180 V=166.7  +MOVJ EC00180
SREFP 3 C00181 BC00181  +REFP EC00181
CALL JOB:SEARCH-R1-S13D
SET P034 P006
SFTON3D P034
SMOVL C00182 BC00182 V=166.7  +MOVJ EC00182
SMOVL C00183 BC00183 V=166.7  +MOVJ EC00183
SREFP 3 C00184 BC00184  +REFP EC00184
CALL JOB:SEARCH-R1-S13D
SET P034 P006
SFTON3D P034
SMOVL C00185 BC00185 V=166.7  +MOVJ EC00185
SFTOF3D
SMOVL C00186 BC00186 V=166.7  +MOVJ EC00186
SREFP 3 C00187 BC00187  +REFP EC00187
CALL JOB:SEARCH-R1-S13D
SET P057 P006
SFTON3D P057
SMOVL C00188 BC00188 V=166.7  +MOVJ EC00188
SREFP 3 C00189 BC00189  +REFP EC00189
CALL JOB:SEARCH-R1-S13D
SET P057 P006
SFTON3D P057
SMOVL C00190 BC00190 V=166.7  +MOVJ EC00190
SFTOF3D
SMOVL C00191 BC00191 V=666.7  +MOVJ EC00191
SMOVL C00192 BC00192 V=166.7  +MOVJ EC00192
SREFP 3 C00193 BC00193  +REFP EC00193
CALL JOB:SEARCH-R1-S13D
SET P058 P006
SFTON3D P058
SMOVL C00194 BC00194 V=166.7  +MOVJ EC00194
SREFP 3 C00195 BC00195  +REFP EC00195
CALL JOB:SEARCH-R1-S13D
SET P058 P006
SFTON3D P058
SFTOF3D
SMOVL C00196 BC00196 V=166.7  +MOVJ EC00196
SMOVL C00197 BC00197 V=666.7  +MOVJ EC00197
SMOVL C00198 BC00198 V=166.7  +MOVJ EC00198
SREFP 3 C00199 BC00199  +REFP EC00199
CALL JOB:SEARCH-R1-S13D
SET P059 P006
SFTON3D P059
SMOVL C00200 BC00200 V=166.7  +MOVJ EC00200
SREFP 3 C00201 BC00201  +REFP EC00201
CALL JOB:SEARCH-R1-S13D
SET P059 P006
SFTON3D P059
SFTOF3D
SMOVL C00202 BC00202 V=166.7  +MOVJ EC00202
SMOVL C00203 BC00203 V=666.7  +MOVJ EC00203
SMOVL C00204 BC00204 V=500.0  +MOVJ EC00204
SMOVL C00205 BC00205 V=166.7  +MOVJ EC00205
SREFP 3 C00206 BC00206  +REFP EC00206
CALL JOB:SEARCH-R1-S13D
SET P060 P006
SFTON3D P060
SMOVL C00207 BC00207 V=166.7  +MOVJ EC00207
SREFP 3 C00208 BC00208  +REFP EC00208
CALL JOB:SEARCH-R1-S13D
SET P060 P006
SFTON3D P060
SMOVL C00209 BC00209 V=166.7  +MOVJ EC00209
SFTOF3D
MOVJ C00210 BC00210 VJ=100.00  +MOVJ EC00210 VJ=100.00
MOVJ C00211 BC00211 VJ=100.00  +MOVJ EC00211 VJ=100.00
MOVJ C00212 BC00212 VJ=100.00  +MOVJ EC00212 VJ=100.00
MOVJ C00213 BC00213 VJ=100.00  +MOVJ EC00213 VJ=100.00
SMOVL C00214 BC00214 V=166.7  +MOVJ EC00214
SREFP 3 C00215 BC00215  +REFP EC00215
CALL JOB:SEARCH-R1-S13D
SET P090 P006
SFTON3D P090
SMOVL C00216 BC00216 V=166.7  +MOVJ EC00216
SREFP 3 C00217 BC00217  +REFP EC00217
CALL JOB:SEARCH-R1-S13D
SET P090 P006
SFTON3D P090
SMOVL C00218 BC00218 V=166.7  +MOVJ EC00218
SFTOF3D
SMOVL C00219 BC00219 V=666.7  +MOVJ EC00219
SMOVL C00220 BC00220 V=166.7  +MOVJ EC00220
SREFP 3 C00221 BC00221  +REFP EC00221
CALL JOB:SEARCH-R1-S13D
SET P091 P006
SFTON3D P091
SMOVL C00222 BC00222 V=166.7  +MOVJ EC00222
SREFP 3 C00223 BC00223  +REFP EC00223
CALL JOB:SEARCH-R1-S13D
SET P091 P006
SFTON3D P091
SMOVL C00224 BC00224 V=166.7  +MOVJ EC00224
MACRO1 MJ#(0) ARGF6
SMOVL C00225 BC00225 V=166.7  +MOVJ EC00225
ARCON
SFTON3D P090
SMOVL C00226 BC00226 V=11.7  +MOVJ EC00226
ARCOF
SFTOF3D
SMOVL C00227 BC00227 V=166.7  +MOVJ EC00227
MOVJ C00228 BC00228 VJ=100.00  +MOVJ EC00228 VJ=100.00
MOVJ C00229 BC00229 VJ=100.00  +MOVJ EC00229 VJ=100.00
'
MOVJ C00230 BC00230 VJ=100.00  +MOVJ EC00230 VJ=100.00
'Path W3658
SFTOF3D
SFTON3D P039
MOVJ C00231 BC00231 VJ=100.00  +MOVJ EC00231 VJ=100.00
MACRO1 MJ#(0) ARGF14
SFTOF3D
SFTON3D P039
SMOVL C00232 BC00232 V=133.3  +MOVJ EC00232
SREFP 1 C00233 BC00233  +REFP EC00233
SREFP 2 C00234 BC00234  +REFP EC00234
MACRO1 MJ#(0) ARGF14
ARCON
SMOVL C00235 BC00235 V=10.0  +MOVJ EC00235
SMOVL C00236 BC00236 V=10.0  +MOVJ EC00236
SMOVL C00237 BC00237 V=11.7  +MOVJ EC00237
SMOVL C00238 BC00238 V=11.7  +MOVJ EC00238
SMOVL C00239 BC00239 V=11.7  +MOVJ EC00239
ARCOF
'Path W3659
SFTOF3D
MOVJ C00240 BC00240 VJ=25.00  +MOVJ EC00240 VJ=100.00
MOVJ C00241 BC00241 VJ=100.00  +MOVJ EC00241 VJ=100.00
'Path W3661
SFTOF3D
SFTON3D P038
MOVJ C00242 BC00242 VJ=100.00  +MOVJ EC00242 VJ=100.00
SMOVL C00243 BC00243 V=500.0  +MOVJ EC00243
SMOVL C00244 BC00244 V=133.3 PL=0  +MOVJ EC00244
SREFP 1 C00245 BC00245  +REFP EC00245
SREFP 2 C00246 BC00246  +REFP EC00246
ARCON
SMOVL C00247 BC00247 V=9.2  +MOVJ EC00247
SMOVL C00248 BC00248 V=9.2  +MOVJ EC00248
ARCOF
SMOVL C00249 BC00249 V=400.0  +MOVJ EC00249
SMOVL C00250 BC00250 V=1000.0  +MOVJ EC00250
SFTOF3D
'Path W3662
SFTOF3D
SFTON3D P038
MOVJ C00251 BC00251 VJ=100.00  +MOVJ EC00251 VJ=100.00
SMOVL C00252 BC00252 V=400.0  +MOVJ EC00252
SMOVL C00253 BC00253 V=133.3 PL=0  +MOVJ EC00253
SREFP 1 C00254 BC00254  +REFP EC00254
SREFP 2 C00255 BC00255  +REFP EC00255
ARCON
SMOVL C00256 BC00256 V=10.0  +MOVJ EC00256
SMOVL C00257 BC00257 V=10.0  +MOVJ EC00257
SMOVL C00258 BC00258 V=10.0  +MOVJ EC00258
ARCOF
SMOVL C00259 BC00259 V=400.0  +MOVJ EC00259
SMOVL C00260 BC00260 V=1000.0  +MOVJ EC00260
SFTOF3D
'Path W3663
SFTOF3D
SFTON3D P038
SMOVL C00261 BC00261 V=666.7  +MOVJ EC00261
SMOVL C00262 BC00262 V=100.0 PL=0  +MOVJ EC00262
SREFP 1 C00263 BC00263  +REFP EC00263
SREFP 2 C00264 BC00264  +REFP EC00264
ARCON
SMOVL C00265 BC00265 V=10.0  +MOVJ EC00265
SMOVL C00266 BC00266 V=10.0  +MOVJ EC00266
SMOVL C00267 BC00267 V=10.0  +MOVJ EC00267
ARCOF
SMOVL C00268 BC00268 V=400.0  +MOVJ EC00268
SFTOF3D
MOVJ C00269 BC00269 VJ=100.00  +MOVJ EC00269 VJ=100.00
'Path W3664
SFTOF3D
SFTON3D P033
MOVJ C00270 BC00270 VJ=100.00  +MOVJ EC00270 VJ=100.00
SMOVL C00271 BC00271 V=666.7  +MOVJ EC00271
SMOVL C00272 BC00272 V=666.7  +MOVJ EC00272
SMOVL C00273 BC00273 V=133.3 PL=0  +MOVJ EC00273
SREFP 1 C00274 BC00274  +REFP EC00274
SREFP 2 C00275 BC00275  +REFP EC00275
MACRO1 MJ#(0) ARGF14
ARCON
SMOVL C00276 BC00276 V=9.2  +MOVJ EC00276
SMOVL C00277 BC00277 V=9.2  +MOVJ EC00277
SMOVL C00278 BC00278 V=9.2  +MOVJ EC00278
SMOVL C00279 BC00279 V=9.2  +MOVJ EC00279
SMOVL C00280 BC00280 V=9.2  +MOVJ EC00280
SMOVL C00281 BC00281 V=9.2  +MOVJ EC00281
ARCOF
SMOVL C00282 BC00282 V=400.0  +MOVJ EC00282
SMOVL C00283 BC00283 V=1000.0  +MOVJ EC00283
SFTOF3D
'Path W3666
SFTOF3D
SFTON3D P033
SMOVL C00284 BC00284 V=133.3 PL=0  +MOVJ EC00284
SREFP 1 C00285 BC00285  +REFP EC00285
SREFP 2 C00286 BC00286  +REFP EC00286
MACRO1 MJ#(0) ARGF14
ARCON
SMOVL C00287 BC00287 V=10.0  +MOVJ EC00287
SMOVL C00288 BC00288 V=10.0  +MOVJ EC00288
ARCOF
SMOVL C00289 BC00289 V=400.0  +MOVJ EC00289
SFTOF3D
MOVJ C00290 BC00290 VJ=80.00  +MOVJ EC00290 VJ=50.00
'12
'Path W3667
SFTOF3D
SFTON3D P034
MOVJ C00291 BC00291 VJ=100.00  +MOVJ EC00291 VJ=100.00
SMOVL C00292 BC00292 V=666.7  +MOVJ EC00292
SFTON3D P034
SMOVL C00293 BC00293 V=133.3 PL=0  +MOVJ EC00293
SREFP 1 C00294 BC00294  +REFP EC00294
SREFP 2 C00295 BC00295  +REFP EC00295
MACRO1 MJ#(0) ARGF6
ARCON
SWVON WEV#(21)
SMOVL C00296 BC00296 V=10.0  +MOVJ EC00296
SMOVL C00297 BC00297 V=10.0  +MOVJ EC00297
SMOVL C00298 BC00298 V=10.0  +MOVJ EC00298
ARCOF
SWVOF
SFTOF3D
SMOVL C00299 BC00299 V=400.0  +MOVJ EC00299
MOVJ C00300 BC00300 VJ=100.00  +MOVJ EC00300 VJ=15.00
'Path W3668
SFTOF3D
SFTON3D P036
MOVJ C00301 BC00301 VJ=100.00  +MOVJ EC00301 VJ=100.00
SMOVL C00302 BC00302 V=666.7  +MOVJ EC00302
SMOVL C00303 BC00303 V=133.3 PL=0  +MOVJ EC00303
SREFP 1 C00304 BC00304  +REFP EC00304
SREFP 2 C00305 BC00305  +REFP EC00305
MACRO1 MJ#(0) ARGF14
ARCON
SMOVL C00306 BC00306 V=9.2  +MOVJ EC00306
SMOVL C00307 BC00307 V=9.2  +MOVJ EC00307
SMOVL C00308 BC00308 V=9.2  +MOVJ EC00308
SMOVL C00309 BC00309 V=9.2  +MOVJ EC00309
ARCOF
SMOVL C00310 BC00310 V=400.0  +MOVJ EC00310
SMOVL C00311 BC00311 V=1000.0  +MOVJ EC00311
MOVJ C00312 BC00312 VJ=100.00  +MOVJ EC00312 VJ=15.00
MOVJ C00313 BC00313 VJ=100.00  +MOVJ EC00313 VJ=15.00
SFTON3D P036
MOVJ C00314 BC00314 VJ=100.00  +MOVJ EC00314 VJ=100.00
SMOVL C00315 BC00315 V=400.0  +MOVJ EC00315
SMOVL C00316 BC00316 V=133.3 PL=0  +MOVJ EC00316
SREFP 1 C00317 BC00317  +REFP EC00317
SREFP 2 C00318 BC00318  +REFP EC00318
MACRO1 MJ#(0) ARGF14
ARCON
SMOVL C00319 BC00319 V=10.0  +MOVJ EC00319
ARCOF
SMOVL C00320 BC00320 V=400.0  +MOVJ EC00320
SMOVL C00321 BC00321 V=1000.0  +MOVJ EC00321
SFTOF3D
'13
MOVJ C00322 BC00322 VJ=100.00  +MOVJ EC00322 VJ=100.00
MOVJ C00323 BC00323 VJ=100.00  +MOVJ EC00323 VJ=100.00
'Path W3671
SFTOF3D
SFTON3D P052
SMOVL C00324 BC00324 V=400.0  +MOVJ EC00324
MACRO1 MJ#(0) ARGF9
SMOVL C00325 BC00325 V=133.3  +MOVJ EC00325
ARCON
SMOVL C00326 BC00326 V=10.8  +MOVJ EC00326
SMOVL C00327 BC00327 V=10.8  +MOVJ EC00327
ARCOF
SMOVL C00328 BC00328 V=166.7  +MOVJ EC00328
SMOVL C00329 BC00329 V=133.3 PL=0  +MOVJ EC00329
SREFP 1 C00330 BC00330  +REFP EC00330
SREFP 2 C00331 BC00331  +REFP EC00331
MACRO1 MJ#(0) ARGF9
ARCON
SMOVL C00332 BC00332 V=10.8  +MOVJ EC00332
SFTON3D P041
SMOVL C00333 BC00333 V=10.8  +MOVJ EC00333
ARCOF
SMOVL C00334 BC00334 V=400.0  +MOVJ EC00334
SFTOF3D
'14
'Path W3672
SFTOF3D
SFTON3D P043
MOVJ C00335 BC00335 VJ=100.00  +MOVJ EC00335 VJ=100.00
MOVJ C00336 BC00336 VJ=100.00  +MOVJ EC00336 VJ=100.00
SMOVL C00337 BC00337 V=1000.0  +MOVJ EC00337
SFTON3D P055
SMOVL C00338 BC00338 V=166.7  +MOVJ EC00338
ARCON
SMOVL C00339 BC00339 V=10.0  +MOVJ EC00339
ARCOF
SFTOF3D
MOVJ C00340 BC00340 VJ=50.00  +MOVJ EC00340 VJ=100.00
MOVJ C00341 BC00341 VJ=100.00  +MOVJ EC00341 VJ=50.00
SFTON3D P056
SMOVL C00342 BC00342 V=250.0  +MOVJ EC00342
SMOVL C00343 BC00343 V=133.3  +MOVJ EC00343
ARCON
SMOVL C00344 BC00344 V=10.0  +MOVJ EC00344
ARCOF
SMOVL C00345 BC00345 V=333.3  +MOVJ EC00345
SFTOF3D
'15-brak
'16
'Path W3673
SFTOF3D
SFTON3D P037
MOVJ C00346 BC00346 VJ=100.00  +MOVJ EC00346 VJ=100.00
SMOVL C00347 BC00347 V=666.7  +MOVJ EC00347
SMOVL C00348 BC00348 V=133.3 PL=0  +MOVJ EC00348
SREFP 1 C00349 BC00349  +REFP EC00349
SREFP 2 C00350 BC00350  +REFP EC00350
MACRO1 MJ#(0) ARGF14
ARCON
SMOVL C00351 BC00351 V=10.0  +MOVJ EC00351
SMOVL C00352 BC00352 V=10.0  +MOVJ EC00352
SMOVL C00353 BC00353 V=10.0  +MOVJ EC00353
ARCOF
SFTOF3D
SFTON3D P037
SMOVL C00354 BC00354 V=166.7 PL=0  +MOVJ EC00354
SREFP 1 C00355 BC00355  +REFP EC00355
SREFP 2 C00356 BC00356  +REFP EC00356
ARCON
SMOVL C00357 BC00357 V=10.0  +MOVJ EC00357
ARCON
SMOVL C00358 BC00358 V=10.0  +MOVJ EC00358
ARCOF
SMOVL C00359 BC00359 V=250.0  +MOVJ EC00359
SMOVL C00360 BC00360 V=400.0  +MOVJ EC00360
SFTOF3D
MOVJ C00361 BC00361 VJ=100.00  +MOVJ EC00361 VJ=100.00
'Path W3675
SFTOF3D
SFTON3D P037
MOVJ C00362 BC00362 VJ=100.00  +MOVJ EC00362 VJ=100.00
SMOVL C00363 BC00363 V=400.0  +MOVJ EC00363
SMOVL C00364 BC00364 V=166.7 PL=0  +MOVJ EC00364
SREFP 1 C00365 BC00365  +REFP EC00365
SREFP 2 C00366 BC00366  +REFP EC00366
ARCON
SMOVL C00367 BC00367 V=10.0  +MOVJ EC00367
SMOVL C00368 BC00368 V=10.0  +MOVJ EC00368
SMOVL C00369 BC00369 V=10.0  +MOVJ EC00369
ARCOF
SMOVL C00370 BC00370 V=400.0  +MOVJ EC00370
SMOVL C00371 BC00371 V=1000.0  +MOVJ EC00371
SFTOF3D
'17
MOVJ C00372 BC00372 VJ=100.00  +MOVJ EC00372 VJ=100.00
'Path W3676
SFTOF3D
SFTON3D P040
MOVJ C00373 BC00373 VJ=100.00  +MOVJ EC00373 VJ=100.00
SMOVL C00374 BC00374 V=400.0  +MOVJ EC00374
SMOVL C00375 BC00375 V=166.7 PL=0  +MOVJ EC00375
SREFP 1 C00376 BC00376  +REFP EC00376
SREFP 2 C00377 BC00377  +REFP EC00377
ARCON
SMOVL C00378 BC00378 V=10.0  +MOVJ EC00378
SMOVL C00379 BC00379 V=10.0  +MOVJ EC00379
SMOVL C00380 BC00380 V=10.0  +MOVJ EC00380
ARCOF
SMOVL C00381 BC00381 V=400.0  +MOVJ EC00381
SMOVL C00382 BC00382 V=1000.0  +MOVJ EC00382
SFTOF3D
'Path W3677
SFTOF3D
SFTON3D P040
SMOVL C00383 BC00383 V=400.0  +MOVJ EC00383
SMOVL C00384 BC00384 V=133.3 PL=0  +MOVJ EC00384
SREFP 1 C00385 BC00385  +REFP EC00385
SREFP 2 C00386 BC00386  +REFP EC00386
ARCON
SMOVL C00387 BC00387 V=10.0  +MOVJ EC00387
SMOVL C00388 BC00388 V=10.0  +MOVJ EC00388
SMOVL C00389 BC00389 V=10.0  +MOVJ EC00389
ARCOF
SMOVL C00390 BC00390 V=400.0  +MOVJ EC00390
MOVJ C00391 BC00391 VJ=100.00  +MOVJ EC00391 VJ=50.00
SFTOF3D
MOVJ C00392 BC00392 VJ=100.00  +MOVJ EC00392 VJ=100.00
'Path W3678
SFTOF3D
SFTON3D P040
SFTOF3D
MOVJ C00393 BC00393 VJ=100.00  +MOVJ EC00393 VJ=100.00
SMOVL C00394 BC00394 V=400.0  +MOVJ EC00394
SMOVL C00395 BC00395 V=133.3 PL=0  +MOVJ EC00395
SREFP 1 C00396 BC00396  +REFP EC00396
SREFP 2 C00397 BC00397  +REFP EC00397
MACRO1 MJ#(0) ARGF14
SMOVL C00398 BC00398 V=25.0  +MOVJ EC00398
ARCOF
SMOVL C00399 BC00399 V=400.0  +MOVJ EC00399
SMOVL C00400 BC00400 V=1000.0  +MOVJ EC00400
SFTOF3D
'18
MOVJ C00401 BC00401 VJ=100.00  +MOVJ EC00401 VJ=100.00
'Path W3679
SFTOF3D
SFTOF3D
SFTON3D P032
MOVJ C00402 BC00402 VJ=100.00  +MOVJ EC00402 VJ=100.00
SMOVL C00403 BC00403 V=400.0  +MOVJ EC00403
SMOVL C00404 BC00404 V=166.7  +MOVJ EC00404
SREFP 1 C00405 BC00405  +REFP EC00405
SREFP 2 C00406 BC00406  +REFP EC00406
MACRO1 MJ#(0) ARGF14
ARCON
SMOVL C00407 BC00407 V=9.2  +MOVJ EC00407
SMOVL C00408 BC00408 V=9.2  +MOVJ EC00408
SMOVL C00409 BC00409 V=9.2  +MOVJ EC00409
SMOVL C00410 BC00410 V=9.2  +MOVJ EC00410
SMOVL C00411 BC00411 V=9.2  +MOVJ EC00411
ARCOF
SMOVL C00412 BC00412 V=400.0  +MOVJ EC00412
SFTOF3D
'Path W3680
SMOVL C00413 BC00413 V=1000.0  +MOVJ EC00413
SFTOF3D
'19
MOVJ C00414 BC00414 VJ=100.00  +MOVJ EC00414 VJ=70.00
'Path W3681
SFTOF3D
SFTON3D P035
MOVJ C00415 BC00415 VJ=100.00  +MOVJ EC00415 VJ=100.00
SMOVL C00416 BC00416 V=400.0  +MOVJ EC00416
SMOVL C00417 BC00417 V=133.3 PL=0  +MOVJ EC00417
SREFP 1 C00418 BC00418  +REFP EC00418
SREFP 2 C00419 BC00419  +REFP EC00419
MACRO1 MJ#(0) ARGF6
ARCON
SWVON WEV#(21)
SMOVL C00420 BC00420 V=9.2  +MOVJ EC00420
ARCOF
SWVOF
SMOVL C00421 BC00421 V=400.0  +MOVJ EC00421
SMOVL C00422 BC00422 V=1000.0  +MOVJ EC00422
SFTOF3D
'20
MOVJ C00423 BC00423 VJ=100.00  +MOVJ EC00423 VJ=100.00
MOVJ C00424 BC00424 VJ=100.00  +MOVJ EC00424 VJ=100.00
'Path W3682
SFTOF3D
SFTON3D P042
SMOVL C00425 BC00425 V=400.0  +MOVJ EC00425
SMOVL C00426 BC00426 V=133.3 PL=0  +MOVJ EC00426
SREFP 1 C00427 BC00427  +REFP EC00427
SREFP 2 C00428 BC00428  +REFP EC00428
MACRO1 MJ#(0) ARGF6
ARCON
SMOVL C00429 BC00429 V=7.5  +MOVJ EC00429
SMOVL C00430 BC00430 V=7.5  +MOVJ EC00430
SMOVL C00431 BC00431 V=7.5  +MOVJ EC00431
ARCOF
SMOVL C00432 BC00432 V=400.0  +MOVJ EC00432
SFTOF3D
SFTON3D P042
SMOVL C00433 BC00433 V=400.0  +MOVJ EC00433
SMOVL C00434 BC00434 V=133.3 PL=0  +MOVJ EC00434
SREFP 1 C00435 BC00435  +REFP EC00435
SREFP 2 C00436 BC00436  +REFP EC00436
MACRO1 MJ#(0) ARGF6
ARCON
SMOVL C00437 BC00437 V=10.0  +MOVJ EC00437
ARCOF
SMOVL C00438 BC00438 V=400.0  +MOVJ EC00438
SMOVL C00439 BC00439 V=1000.0  +MOVJ EC00439
SFTOF3D
'Path W3686
SFTOF3D
SFTON3D P042
MOVJ C00440 BC00440 VJ=100.00  +MOVJ EC00440 VJ=100.00
SMOVL C00441 BC00441 V=400.0  +MOVJ EC00441
SMOVL C00442 BC00442 V=166.7 PL=0  +MOVJ EC00442
SREFP 1 C00443 BC00443  +REFP EC00443
SREFP 2 C00444 BC00444  +REFP EC00444
MACRO1 MJ#(0) ARGF6
ARCON
SMOVL C00445 BC00445 V=10.0  +MOVJ EC00445
ARCOF
SMOVL C00446 BC00446 V=400.0  +MOVJ EC00446
SMOVL C00447 BC00447 V=1000.0  +MOVJ EC00447
SFTOF3D
'21
MOVJ C00448 BC00448 VJ=100.00  +MOVJ EC00448 VJ=100.00
MOVJ C00449 BC00449 VJ=100.00  +MOVJ EC00449 VJ=100.00
MOVJ C00450 BC00450 VJ=70.00  +MOVJ EC00450 VJ=70.00
'Path W3687
SFTOF3D
SFTON3D P031
SMOVL C00451 BC00451 V=833.3  +MOVJ EC00451
SMOVL C00452 BC00452 V=166.7 PL=0  +MOVJ EC00452
SREFP 1 C00453 BC00453  +REFP EC00453
SREFP 2 C00454 BC00454  +REFP EC00454
MACRO1 MJ#(0) ARGF9
ARCON
SMOVL C00455 BC00455 V=10.8  +MOVJ EC00455
SFTON3D P051
SMOVL C00456 BC00456 V=12.5  +MOVJ EC00456
SMOVL C00457 BC00457 V=12.5  +MOVJ EC00457
SMOVL C00458 BC00458 V=12.5  +MOVJ EC00458
ARCOF
SMOVL C00459 BC00459 V=400.0  +MOVJ EC00459
MOVJ C00460 BC00460 VJ=100.00  +MOVJ EC00460 VJ=50.00
MOVJ C00461 BC00461 VJ=100.00  +MOVJ EC00461 VJ=50.00
MACRO1 MJ#(0) ARGF14
MOVJ C00462 BC00462 VJ=100.00  +MOVJ EC00462 VJ=100.00
SFTON3D P034
SMOVL C00463 BC00463 V=166.7  +MOVJ EC00463
ARCON
SMOVL C00464 BC00464 V=10.0  +MOVJ EC00464
ARCOF
SMOVL C00465 BC00465 V=166.7  +MOVJ EC00465
SFTOF3D
SMOVL C00466 BC00466 V=333.3  +MOVJ EC00466
SFTOF3D
MACRO1 MJ#(0) ARGF9
SFTON3D P058
SMOVL C00467 BC00467 V=166.7  +MOVJ EC00467
ARCON
SMOVL C00468 BC00468 V=11.7  +MOVJ EC00468
ARCOF
SMOVL C00469 BC00469 V=333.3  +MOVJ EC00469
SFTOF3D
SMOVL C00470 BC00470 V=333.3  +MOVJ EC00470
MACRO1 MJ#(0) ARGF9
SFTON3D P057
SMOVL C00471 BC00471 V=166.7 PL=0  +MOVJ EC00471
ARCON
SMOVL C00472 BC00472 V=9.2  +MOVJ EC00472
SFTON3D P058
SMOVL C00473 BC00473 V=9.2  +MOVJ EC00473
SFTON3D P059
SWVON WEV#(30)
SMOVL C00474 BC00474 V=8.7  +MOVJ EC00474
SMOVL C00475 BC00475 V=8.7  +MOVJ EC00475
SMOVL C00476 BC00476 V=8.7  +MOVJ EC00476
ARCOF
SWVOF
SFTOF3D
SMOVL C00477 BC00477 V=250.0  +MOVJ EC00477
MOVJ C00478 BC00478 VJ=100.00  +MOVJ EC00478 VJ=100.00
MOVJ C00479 BC00479 VJ=100.00  +MOVJ EC00479 VJ=100.00
SFTON3D P060
SREFP 1 C00480 BC00480  +REFP EC00480
SREFP 2 C00481 BC00481  +REFP EC00481
SMOVL C00482 BC00482 V=250.0  +MOVJ EC00482
ARCON
SWVON WEV#(12)
SMOVL C00483 BC00483 V=10.0  +MOVJ EC00483
ARCOF
SWVOF
SMOVL C00484 BC00484 V=250.0  +MOVJ EC00484
SFTOF3D
MOVJ C00485 BC00485 VJ=100.00  +MOVJ EC00485 VJ=100.00
MOVJ C00486 BC00486 VJ=100.00  +MOVJ EC00486 VJ=70.00
CALL JOB:CLEAN-R1_KM_NEW
MOVJ C00487 BC00487 VJ=100.00  +MOVJ EC00487 VJ=100.00
'cut_wire_dol
'Path S3688
SFTOF3D
MOVJ C00488 BC00488 VJ=100.00  +MOVJ EC00488 VJ=70.00
MOVJ C00489 BC00489 VJ=100.00  +MOVJ EC00489 VJ=70.00
MOVJ C00490 BC00490 VJ=100.00  +MOVJ EC00490 VJ=100.00
MOVL C00491 BC00491 V=400.0  +MOVJ EC00491 VJ=100.00
SMOVL C00492 BC00492 V=100.0  +MOVJ EC00492
SREFP 3 C00493 BC00493  +REFP EC00493
CALL JOB:SEARCH-R1-S13D
SET P023 P006
SFTON3D P023
SMOVL C00494 BC00494 V=100.0  +MOVJ EC00494
SREFP 3 C00495 BC00495  +REFP EC00495
CALL JOB:SEARCH-R1-S13D
SET P023 P006
SFTON3D P023
SMOVL C00496 BC00496 V=100.0  +MOVJ EC00496
MOVL C00497 BC00497 V=400.0  +MOVJ EC00497 VJ=100.00
MOVL C00498 BC00498 V=1000.0  +MOVJ EC00498 VJ=100.00
MOVJ C00499 BC00499 VJ=100.00  +MOVJ EC00499 VJ=100.00
'Path S3689
SFTOF3D
MOVJ C00500 BC00500 VJ=100.00  +MOVJ EC00500 VJ=100.00
MOVL C00501 BC00501 V=400.0  +MOVJ EC00501 VJ=100.00
SMOVL C00502 BC00502 V=100.0  +MOVJ EC00502
SREFP 3 C00503 BC00503  +REFP EC00503
CALL JOB:SEARCH-R1-S13D
SET P022 P006
SFTON3D P022
SMOVL C00504 BC00504 V=100.0  +MOVJ EC00504
SREFP 3 C00505 BC00505  +REFP EC00505
CALL JOB:SEARCH-R1-S13D
SET P022 P006
SFTON3D P022
SMOVL C00506 BC00506 V=250.0  +MOVJ EC00506
SFTOF3D
SMOVL C00507 BC00507 V=1000.0  +MOVJ EC00507
SMOVL C00508 BC00508 V=1000.0  +MOVJ EC00508
SMOVL C00509 BC00509 V=1000.0  +MOVJ EC00509
SMOVL C00510 BC00510 V=333.3  +MOVJ EC00510
SREFP 3 C00511 BC00511  +REFP EC00511
CALL JOB:SEARCH-R1-S13D
SET P060 P006
SFTON3D P060
SMOVL C00512 BC00512 V=166.7  +MOVJ EC00512
SMOVL C00513 BC00513 V=166.7  +MOVJ EC00513
SREFP 3 C00514 BC00514  +REFP EC00514
CALL JOB:SEARCH-R1-S13D
SET P060 P006
SFTON3D P060
SMOVL C00515 BC00515 V=166.7  +MOVJ EC00515
MOVJ C00516 BC00516 VJ=15.00  +MOVJ EC00516 VJ=0.78
MOVJ C00517 BC00517 VJ=15.00  +MOVJ EC00517 VJ=15.00
SMOVL C00518 BC00518 V=166.7  +MOVJ EC00518
SREFP 3 C00519 BC00519  +REFP EC00519
CALL JOB:SEARCH-R1-S13D
SET P060 P006
SFTON3D P060
SMOVL C00520 BC00520 V=416.7  +MOVJ EC00520
SFTOF3D
SMOVL C00521 BC00521 V=416.7  +MOVJ EC00521
SMOVL C00522 BC00522 V=416.7  +MOVJ EC00522
SREFP 3 C00523 BC00523  +REFP EC00523
CALL JOB:SEARCH-R1-S13D
SET P061 P006
SFTON3D P061
SMOVL C00524 BC00524 V=166.7  +MOVJ EC00524
SREFP 3 C00525 BC00525  +REFP EC00525
CALL JOB:SEARCH-R1-S13D
SET P061 P006
SFTON3D P061
SMOVL C00526 BC00526 V=500.0  +MOVJ EC00526
SMOVL C00527 BC00527 V=500.0  +MOVJ EC00527
SMOVL C00528 BC00528 V=1000.0  +MOVJ EC00528
MOVJ C00529 BC00529 VJ=100.00  +MOVJ EC00529 VJ=100.00
MOVJ C00530 BC00530 VJ=100.00  +MOVJ EC00530 VJ=100.00
MOVJ C00531 BC00531 VJ=100.00  +MOVJ EC00531 VJ=100.00
'Path S3690
SFTOF3D
MOVJ C00532 BC00532 VJ=100.00  +MOVJ EC00532 VJ=100.00
MOVL C00533 BC00533 V=400.0  +MOVJ EC00533 VJ=100.00
SMOVL C00534 BC00534 V=100.0  +MOVJ EC00534
SREFP 3 C00535 BC00535  +REFP EC00535
CALL JOB:SEARCH-R1-S13D
SET P021 P006
SFTON3D P021
SMOVL C00536 BC00536 V=100.0  +MOVJ EC00536
SREFP 3 C00537 BC00537  +REFP EC00537
CALL JOB:SEARCH-R1-S13D
SET P021 P006
